			IF CIR_STOP_REQ THEN Pump_En[2] := 1;
			ELSIF CIR_RUN_REQ THEN Pump_En[2] := 0;
			ELSE Pump_En[2] := BOOL_TO_WORD(NOT Delay.OUT);
			END_IF

			(* Set RUN signal (for external objects) *)
			IF AlarmCtr>0 THEN (*OR fPump_ST[1].OUT OR fPump_ST[2].OUT THEN*)
				Run:=FALSE;
			ELSE
				Run:=SEL(Pump_En[2]=1,FALSE,TRUE);
			END_IF
		END_IF


	1,2:  (*** Alternate working and Master/backup mode ***)
		IF fCIR_AUTO[ActivePump].IN THEN
			(* If priority request *)
			IF CIR_STOP_REQ THEN Pump_En[ActivePump] := 1;
			ELSIF CIR_RUN_REQ THEN Pump_En[ActivePump] := 0;
			ELSE Pump_En[ActivePump] := BOOL_TO_WORD(NOT Delay.OUT);
			END_IF

			fBackup(IN:=(AlarmHw[ActivePump].OUT));

			IF fBackup.EVH THEN
				ActivePump := SEL(ActivePump=1,1,2);
				LogEv(EL_Wrn,EO_CIRD,ID,16,'');	(* Pump switched because of current pump failure *)

				(* Switch off old active pump *)
				IF ActivePump=1 THEN Pump_En[2] := 1;
				ELSE Pump_En[1] := 1;
				END_IF
			END_IF


			(* Set RUN signal (for external objects) *)
			IF AlarmCtr>0 THEN (*OR fPump_ST[ActivePump].OUT THEN*)
				Run:=FALSE;
			ELSE
				IF (ActivePump=1 AND PumpB_AUTO) OR (ActivePump=2 AND PumpA_AUTO) THEN
					Run:=SEL(Pump_En[ActivePump]=1,TRUE,FALSE);
				END_IF
			END_IF

		END_IF

END_CASE

(* Check if a pump enable update (modbus write) is requested *)
fPump_En[1](IN:=(Pump_En[1]=1));
fPump_En[2](IN:=(Pump_En[2]=1));

IF fPump_En[1].EVH OR fPump_En[1].EVL THEN
	Refresh_Now := TRUE;
END_IF

IF fPump_En[2].EVH OR fPump_En[2].EVL THEN
	Refresh_Now := TRUE;
END_IF
END_ACTION
ACTION Stm:
CASE state OF
	0:	(* Refresh time manager *)
		ReadTmr(IN:=NOT ReadTmr.Q);
		TimeOutModBus(In:=state<>0,PT:=t#5s);
		IF (ReadTmr.Q AND NodoDaInterrogare=Address1 )OR Refresh_Now AND NOT InibiscoModbus THEN
			state := 10;
			ReadTmr.PT := T#10s;  (* moreno *)
			InibiscoModbus := TRUE;
			Refresh_Now := FALSE;
		END_IF

	(**** READ CIR PARAMETERS ****)

	(**** PUMP 1 ****)
	10:	(* richiedo lettura stato Pompa  *)

			Modbus.MB_Query.SlaveAddress := Address1;
			Modbus.MB_Query.FunctionCode := 3;
			ModBus.MB_Query.Read_StartAddress := 201;
			ModBus.MB_Query.Read_Quantity := 2;
			ModBus.MB_Start := TRUE;

			state := 20;

	20:	(* Ripsosta *)
		IF NOT ModBus.MB_Start   THEN

			VerificaFuctionCode:=ModBus.MB_Resp.FunctionCode;
			VerificaNodoLetto:=ModBus.MB_Resp.SlaveAddress;
			IF ModBus.MB_MASTER.MB_Error<>0 THEN
				state := 45;
			ELSE
				DataPump1.PumpStatus := ModBus.MB_Resp.Data[0];
				DataPump1.PumpFault	:= WORD_TO_BOOL(ModBus.MB_Resp.Data[1]);

				Modbus.MB_Query.SlaveAddress := Address1;
				Modbus.MB_Query.FunctionCode := 3;
				ModBus.MB_Query.Read_StartAddress := 210;
				ModBus.MB_Query.Read_Quantity := 12;
				ModBus.MB_Start := TRUE;

				state := 30;
			END_IF
		END_IF

	30: (* Ripsota Altri paramenti Stato Pompa *)
		IF NOT ModBus.MB_Start  THEN

			IF ModBus.MB_MASTER.MB_Error<>0 THEN (*OR ModBus.MB_MASTER.MB_Error<>0 THEN*)
				state := 45;
			ELSE
				DataPump1.PumpBoardTemp 	:= WORD_TO_INT(ModBus.MB_Resp.Data[0]);
				DataPump1.PumpVoltage	:= ModBus.MB_Resp.Data[2];
				DataPump1.PumpCurrent	:= ModBus.MB_Resp.Data[3];
				DataPump1.PumpRPM		:= ModBus.MB_Resp.Data[5];
				DataPump1.PumpPower		:= ModBus.MB_Resp.Data[6];
				DataPump1.PumpOpTime		:= BUILD_16TO32(ADR(ModBus.MB_Resp.Data[7]));
				DataPump1.PumpHead		:= ModBus.MB_Resp.Data[9];
				DataPump1.PumpFlow		:= ModBus.MB_Resp.Data[10];
				DataPump1.PumpLiqTemp	:= WORD_TO_INT(ModBus.MB_Resp.Data[11]);


				ModBus.MB_Query.Read_StartAddress := 230; (* Lettura Allarmi presenti nella pompa *)
				ModBus.MB_Query.Read_Quantity := 1;(*15;*)
				ModBus.MB_Start := TRUE;

				state := 40;
			END_IF
		END_IF

	40:	(* Read alarms *)
		IF NOT ModBus.MB_Start   THEN
			IF ModBus.MB_MASTER.MB_Error<>0 THEN (*OR ModBus.MB_MASTER.MB_Error<>0 THEN*)
				state := 45;
			ELSE
				DataPump1.PumpAlarm[0] := ModBus.MB_Resp.Data[0];	(* Read just last (most recent) alarm *)
				(*DataPump.PumpAlarm[1] := ModBus.MB_Resp.Data[1];
				DataPump.PumpAlarm[2] := ModBus.MB_Resp.Data[2];
				DataPump.PumpAlarm[3] := ModBus.MB_Resp.Data[3];
				DataPump.PumpAlarm[4] := ModBus.MB_Resp.Data[4];
				DataPump.PumpAlarm[5] := ModBus.MB_Resp.Data[5];
				DataPump.PumpAlarm[6] := ModBus.MB_Resp.Data[6];
				DataPump.PumpAlarm[7] := ModBus.MB_Resp.Data[7];
				DataPump.PumpAlarm[8] := ModBus.MB_Resp.Data[8];
				DataPump.PumpAlarm[9] := ModBus.MB_Resp.Data[9];
				DataPump.PumpAlarm[10] := ModBus.MB_Resp.Data[10];
				DataPump.PumpAlarm[11] := ModBus.MB_Resp.Data[11];
				DataPump.PumpAlarm[12] := ModBus.MB_Resp.Data[12];
				DataPump.PumpAlarm[13] := ModBus.MB_Resp.Data[13];
				DataPump.PumpAlarm[14] := ModBus.MB_Resp.Data[14];*)

				state := 41;

			END_IF
		END_IF

(**** Dopo La Lettura Scrivo i paramentri ON/OFF e la velocità  ****)
	 41:	(* Scrivo il comando alla pompa A *)

		Modbus.MB_Query.SlaveAddress := Address1;
		Modbus.MB_Query.FunctionCode := 16;
		ModBus.MB_Query.Write_StartAddress := 109;
		ModBus.MB_Query.Write_Quantity :=2;
		ModBus.MB_Query.Write_Data[0] := VelocitaRichiesta;
		ModBus.MB_Query.Write_Data[1] := Pump_En[1];
		ModBus.MB_Start := TRUE;

		state := 42;

	42:	(* Read alarms *)
		IF NOT ModBus.MB_Start   THEN
			IF ModBus.MB_MASTER.MB_Error<>0 THEN (*OR ModBus.MB_MASTER.MB_Error<>0 THEN*)
				state := 45;
			ELSE
				state := 50;
			END_IF
		END_IF


	(**** CHECK MODBUS ERROR ****)
	45: 	(* Release MODBUS *)
			MODBUS.MB_Lock:=FALSE;

			(* Retries *)
			retry:=retry+1;
			IF retry>3 THEN
				retry:=0;
				(* Verify if slave is dead *)
				IF retryErr < retryErrMaX THEN
					retryErr := retryErr + 1;
				ELSE
					fModbusAlr := TRUE;
					(* Verify ModBus error	*)

					IF fModbusAlr AND ErroreComuModBus1=FALSE THEN
						LogEv(EL_Alarm,EO_CIRDM,ID,13,CONCAT('ErroreModbus_',INT_TO_STRING(ModBus.MB_MASTER.MB_Error)));
						ErroreComuModBus1 := TRUE;
					END_IF
					IF fModbusAlr=FALSE AND retryErr=0 THEN
						LogEv(EL_Log,EO_CIRDM,ID,14,'ComunicazioneModBus_OK');
							ErroreComuModBus1 := FALSE;
					(*	WarningCtr := SEL(WarningCtr=0, WarningCtr-1, 0); *)
					END_IF
				END_IF
				Refresh_Now := FALSE;
			END_IF

			state:=50;



	(**** PUMP 2 ****)
	50:	(* richiedo lettura stato Pompa  *)

			Modbus.MB_Query.SlaveAddress := Address2;
			Modbus.MB_Query.FunctionCode := 3;
			ModBus.MB_Query.Read_StartAddress := 201;
			ModBus.MB_Query.Read_Quantity := 2;
			ModBus.MB_Start := TRUE;

			state := 60;

	60:	(* Ripsosta *)
		IF NOT ModBus.MB_Start   THEN

			VerificaFuctionCode:=ModBus.MB_Resp.FunctionCode;
			VerificaNodoLetto:=ModBus.MB_Resp.SlaveAddress;
			IF ModBus.MB_MASTER.MB_Error<>0 THEN
				state := 300;
			ELSE
				DataPump2.PumpStatus := ModBus.MB_Resp.Data[0];
				DataPump2.PumpFault	:= WORD_TO_BOOL(ModBus.MB_Resp.Data[1]);

				Modbus.MB_Query.SlaveAddress := Address2;
				Modbus.MB_Query.FunctionCode := 3;
				ModBus.MB_Query.Read_StartAddress := 210;
				ModBus.MB_Query.Read_Quantity := 12;
				ModBus.MB_Start := TRUE;

				state := 70;
			END_IF
		END_IF

	70: (* Ripsota Altri paramenti Stato Pompa *)
		IF NOT ModBus.MB_Start  THEN

			IF ModBus.MB_MASTER.MB_Error<>0 THEN (*OR ModBus.MB_MASTER.MB_Error<>0 THEN*)
				state := 300;
			ELSE
				DataPump2.PumpBoardTemp 	:= WORD_TO_INT(ModBus.MB_Resp.Data[0]);
				DataPump2.PumpVoltage	:= ModBus.MB_Resp.Data[2];
				DataPump2.PumpCurrent	:= ModBus.MB_Resp.Data[3];
				DataPump2.PumpRPM		:= ModBus.MB_Resp.Data[5];
				DataPump2.PumpPower		:= ModBus.MB_Resp.Data[6];
				DataPump2.PumpOpTime		:= BUILD_16TO32(ADR(ModBus.MB_Resp.Data[7]));
				DataPump2.PumpHead		:= ModBus.MB_Resp.Data[9];
				DataPump2.PumpFlow		:= ModBus.MB_Resp.Data[10];
				DataPump2.PumpLiqTemp	:= WORD_TO_INT(ModBus.MB_Resp.Data[11]);


				ModBus.MB_Query.Read_StartAddress := 230; (* Lettura Allarmi presenti nella pompa *)
				ModBus.MB_Query.Read_Quantity := 1;(*15;*)
				ModBus.MB_Start := TRUE;

				state := 80;
			END_IF
		END_IF

	80:	(* Read alarms *)
		IF NOT ModBus.MB_Start   THEN
			IF ModBus.MB_MASTER.MB_Error<>0 THEN (*OR ModBus.MB_MASTER.MB_Error<>0 THEN*)
				state := 300;
			ELSE
				DataPump2.PumpAlarm[0] := ModBus.MB_Resp.Data[0];	(* Read just last (most recent) alarm *)
				(*DataPump.PumpAlarm[1] := ModBus.MB_Resp.Data[1];
				DataPump.PumpAlarm[2] := ModBus.MB_Resp.Data[2];
				DataPump.PumpAlarm[3] := ModBus.MB_Resp.Data[3];
				DataPump.PumpAlarm[4] := ModBus.MB_Resp.Data[4];
				DataPump.PumpAlarm[5] := ModBus.MB_Resp.Data[5];
				DataPump.PumpAlarm[6] := ModBus.MB_Resp.Data[6];
				DataPump.PumpAlarm[7] := ModBus.MB_Resp.Data[7];
				DataPump.PumpAlarm[8] := ModBus.MB_Resp.Data[8];
				DataPump.PumpAlarm[9] := ModBus.MB_Resp.Data[9];
				DataPump.PumpAlarm[10] := ModBus.MB_Resp.Data[10];
				DataPump.PumpAlarm[11] := ModBus.MB_Resp.Data[11];
				DataPump.PumpAlarm[12] := ModBus.MB_Resp.Data[12];
				DataPump.PumpAlarm[13] := ModBus.MB_Resp.Data[13];
				DataPump.PumpAlarm[14] := ModBus.MB_Resp.Data[14];*)

				state := 100;

			END_IF
		END_IF


	(**** Dopo La Lettura Scrivo i paramentri ON/OFF e la velocità  ****)
	 100:	(* Scrivo il comando alla pompa A *)

		Modbus.MB_Query.SlaveAddress := Address1;
		Modbus.MB_Query.FunctionCode := 16;
		ModBus.MB_Query.Write_StartAddress := 109;
		ModBus.MB_Query.Write_Quantity :=2;
		ModBus.MB_Query.Write_Data[0] := VelocitaRichiesta;
		ModBus.MB_Query.Write_Data[1] := Pump_En[1];
		ModBus.MB_Start := TRUE;

		state := 110;


		110: (* Scrivo il comando alla pompa B *)
		IF NOT ModBus.MB_Start THEN
			IF ModBus.MB_MASTER.MB_Error<>0 THEN (*OR ModBus.MB_MASTER.MB_Error<>0 THEN*)
				state := 300;
			ELSE
				Modbus.MB_Query.SlaveAddress := Address2;
				Modbus.MB_Query.FunctionCode := 16;
				ModBus.MB_Query.Write_StartAddress := 109;
				ModBus.MB_Query.Write_Quantity :=2;
				ModBus.MB_Query.Write_Data[0] := VelocitaRichiesta;
				ModBus.MB_Query.Write_Data[1] := Pump_En[2];
				ModBus.MB_Start := TRUE;

			state := 120;
			END_IF
		END_IF


		120:
		IF NOT ModBus.MB_Start THEN
			IF ModBus.MB_MASTER.MB_Error<>0 THEN (*OR ModBus.MB_MASTER.MB_Error<>0 THEN*)
				state := 300;
			ELSE
				IF fModbusAlr THEN fModbusAlr := FALSE; END_IF

				NodoDaInterrogare:=Address2+1; (* qui il passo è doppio *)
				InibiscoModbus:=FALSE;
				retryErr := 0;
				retry := 0;
				state := 0;
			END_IF
		END_IF



	(**** CHECK MODBUS ERROR ****)
	300: 	(* Release MODBUS *)
			MODBUS.MB_Lock:=FALSE;

			(* Retries *)
			retry:=retry+1;
			IF retry>3 THEN
				retry:=0;
				(* Verify if slave is dead *)
				IF retryErr < retryErrMaX THEN
					retryErr := retryErr + 1;
				ELSE
					fModbusAlr := TRUE;
					(* Verify ModBus error	*)

					IF fModbusAlr AND ErroreComuModBus2=FALSE THEN
						LogEv(EL_Alarm,EO_CIRDM,ID,13,CONCAT('ErroreModbus_',INT_TO_STRING(ModBus.MB_MASTER.MB_Error)));
						ErroreComuModBus2 := TRUE;
					END_IF
					IF fModbusAlr=FALSE AND retryErr=0 THEN
						LogEv(EL_Log,EO_CIRDM,ID,14,'ComunicazioneModBus_OK');
							ErroreComuModBus2 := FALSE;
					(*	WarningCtr := SEL(WarningCtr=0, WarningCtr-1, 0); *)
					END_IF
				END_IF


				Refresh_Now := FALSE;
			END_IF

			NodoDaInterrogare:=Address2+1; (* qui il passo è doppio *)
			state:=0;
END_CASE



(* Controllo Time Out Ciclo ModBus *)

TimeOutModBus(In:=state<>0,PT:=t#5s);
IF TimeOutModBus.Q THEN
	State:=0;
	Refresh_Now:=TRUE;  (* Rilancio la lettura del nodo *)
	IF MODBUS.MB_Lock=TRUE THEN MODBUS.MB_Lock:=FALSE;END_IF
	IF InibiscoModbus=TRUE THEN InibiscoModbus:=FALSE;END_IF
END_IF
END_ACTION

(* POU Plant_Objects/obj_MODBUS_TCP, ST *)
FUNCTION_BLOCK obj_MODBUS_TCP
(* === MODBUS-TCP PROTOCOL INTERFACE ===
   v1.0[10/06/15] - Create
*)
VAR CONSTANT
	VARS_Max	: BYTE := 32;
END_VAR
VAR_INPUT
	(* Settings *)
	ID			: BYTE;
	IP			: STRING;
	PORT		: WORD:=502;
	(* Interface *)
	MB_MASTER	: ETHERNET_MODBUSMASTER_TCP;
	MB_READBUF	: ARRAY [0..128] OF WORD;
	MB_WRITEBUF : ARRAY [0..128] OF WORD;
	MB_Start	: BOOL;
	MB_Lock		: BOOL;
	(* Variables management *)
	VARS_En		: BOOL;
	VARS		: ARRAY [0..VARS_Max] OF typ_MODBUS_VAR;
	VARS_Check	: BOOL;
	VARS_Alarm	: BOOL;
	(* Variables allocation *)
	VAR_Pointer : POINTER TO ARRAY[0..99] OF WORD;
	VAR_Cfg		: POINTER TO typ_MODBUS_VAR;
END_VAR
VAR_OUTPUT
	(* Status *)
	Status_Log	: BYTE;
	Status_Vis	: DWORD;
END_VAR
VAR
	sta         : BYTE :=0;
	i			: BYTE;
	j			: BYTE;
	Alarm		: FLT_EVENT;

	VarTmr		: TON := (PT:=T#1s);
	VarSta		: BYTE; (* Status *)
	VarCnt		: BYTE; (* Scan counter *)
	VarRetry	: BYTE;
	VarAlarm	: BYTE; (* Last variable with errors *)
END_VAR
MB_MASTER( strIP_ADDRESS:=IP, wPORT:=PORT, tTIME_OUT:=T#750MS, (*xCONNECT:=TRUE,*)
		   ptREAD_DATA:=ADR(MB_READBUF), ptSEND_DATA:=ADR(MB_WRITEBUF), xSEND:=MB_Start );

IF sta=0 THEN
	MB_MASTER.xCONNECT:=TRUE;
	sta:=1;
END_IF

(* Process variable management *)
IF VARS_En THEN VARS_Process(); END_IF

(* Check status *)
Alarm(IN:=(MB_MASTER.wERROR<>0));
IF Alarm.EVH THEN
	LogEv(SEL(MB_MASTER.wERROR>0,EL_Wrn,EL_Alarm),EO_MODBUS_TCP,ID,1,WORD_TO_STRING(MB_MASTER.wERROR));
END_IF
IF Alarm.EVL THEN
	LogEv(EL_Log,EO_MODBUS_TCP,ID,2,'');
END_IF

(* Log/visu status *)
   IF Alarm.IN   THEN Status_Log:=2; Status_Vis:=COLOR_RED;
ELSIF Vars_Alarm THEN Status_Log:=1; Status_Vis:=COLOR_YELLOW;
  				 ELSE Status_Log:=0; Status_Vis:=COLOR_GREEN;
END_IF
END_FUNCTION_BLOCK
ACTION VAR_Search:
(* Search VAR with specific pointer if not found return first free VAR
	[Last VAR is not active... used as safe area...] 
*)
j:=VARS_Max;
FOR i := 0 TO VARS_Max-1 DO
	IF VARS[i].Variable=0 AND j>i THEN j:=i; END_IF
	IF VARS[i].Variable=VAR_Pointer THEN
		VAR_Cfg:=ADR(VARS[i]);
		RETURN;
	END_IF
END_FOR
VAR_Cfg:=ADR(VARS[j]);
END_ACTION
ACTION VARS_Process:
(* Update var timers *)
VarTmr(IN:=(NOT VarTmr.Q));
IF VarTmr.Q THEN
	FOR i := 0 TO VARS_Max DO
		IF VARS[i].Refresh_Cnt>0 THEN VARS[i].Refresh_Cnt:=VARS[i].Refresh_Cnt-1; END_IF
	END_FOR
	VARS_Check:=TRUE;
END_IF


(* Process status *)
CASE VarSta OF
	0: (* === Init *)
		VarCnt:=0;
		VarSta:=1;

	1: (* === Wait check signal *)
		IF VARS_Check THEN
			VARS_Check:=FALSE;
			VarCnt:=0;
			VarSta:=2;
		END_IF

	2: (* === Check loop *)
		IF NOT (MB_Lock OR MB_Start) THEN
			WHILE VarCnt<=(VARS_Max-1) AND VarSta=2 DO
				(* Check only active vars *)
				IF VARS[VarCnt].Variable<>0 THEN
					(* Check var auto-refresh on timer checks *)
					IF VARS[VarCnt].Refresh_Time>0 AND VARS[VarCnt].Refresh_Cnt=0 THEN
						VARS[VarCnt].Refresh_Cnt:=VARS[VarCnt].Refresh_Time;
						VarSta:=3;
					END_IF
					(* Check refresh for change or request *)
					CASE VARS[VarCnt].FunCode OF
						5,6,15,16: (* Write functions *)
							IF VARS[VarCnt].Variable_Size=1 THEN
								IF VARS[VarCnt].Variable^<>VARS[VarCnt].Variable_Mirror THEN
									VARS[VarCnt].Variable_Mirror:=VARS[VarCnt].Variable^;
									VarSta:=3;
								END_IF
							ELSE
								IF VARS[VarCnt].Variable_Mirror<>0 THEN
									VARS[VarCnt].Variable_Mirror:=0;
									VarSta:=3;
								END_IF
							END_IF
						1,2,3,4: (* Write functions *)
							IF VARS[VarCnt].Variable_Mirror<>0 THEN
								VARS[VarCnt].Variable_Mirror:=0;
								VarSta:=3;
							END_IF
					END_CASE
				END_IF
				(* Process query *)
				IF VarSta=3 THEN
					MB_Lock:=TRUE;
					MB_MASTER.bUNIT_ID:=VARS[VarCnt].SlaveAddress;
					MB_MASTER.bFUNCTION_CODE:=VARS[VarCnt].FunCode;
					CASE VARS[VarCnt].FunCode OF
						16#5,16#6,16#F,16#10:
							MB_MASTER.wREAD_ADDRESS:=0;
							MB_MASTER.wREAD_QUANTITY:=0;
							MB_MASTER.wWRITE_ADDRESS:=VARS[VarCnt].FunAddress;
							MB_MASTER.wWRITE_QUANTITY:=VARS[VarCnt].Variable_Size;
							IF VARS[VarCnt].Variable_Size=200 THEN
								COPY_32SWAP16(VARS[VarCnt].Variable, ADR(MB_WRITEBUF));
							ELSIF VARS[VarCnt].Variable_Size>1 THEN
								MEMCPY(VARS[VarCnt].Variable, ADR(MB_WRITEBUF), 2*VARS[VarCnt].Variable_Size);
							ELSE
								MB_WRITEBUF[0]:=VARS[VarCnt].Variable^;
							END_IF
						16#1,16#2,16#3,16#4:
							MB_MASTER.wREAD_ADDRESS:=VARS[VarCnt].FunAddress;
							IF VARS[VarCnt].Variable_Size=200 THEN MB_MASTER.wREAD_QUANTITY:=2; ELSE
							  MB_MASTER.wREAD_QUANTITY:=VARS[VarCnt].Variable_Size;
							END_IF
							MB_MASTER.wWRITE_ADDRESS:=0;
							MB_MASTER.wWRITE_QUANTITY:=0;
					END_CASE
					VarRetry:=0;
					MB_Start:=TRUE;
				ELSE
					VarCnt:=VarCnt+1;
				END_IF
			END_WHILE
			(* Check loop completed -> no actions *)
			IF VarSta=2 THEN VarSta:=1; END_IF
		END_IF

	3: (* === Wait & process MB response *)
		IF NOT MB_Start THEN
			IF MB_MASTER.wERROR=0 THEN
				CASE VARS[VarCnt].FunCode OF
					1,2,3,4:
						IF VARS[VarCnt].Variable_Size=200 THEN
							COPY_32SWAP16(ADR(MB_READBUF), VARS[VarCnt].Variable);
						ELSIF VARS[VarCnt].Variable_Size>1 THEN
							MEMCPY(ADR(MB_READBUF), VARS[VarCnt].Variable, 2*VARS[VarCnt].Variable_Size);
						ELSE
							VARS[VarCnt].Variable^:=MB_READBUF[0];
						END_IF
				END_CASE
				MB_Lock:=FALSE;
				(* Signal error recovery *)
				IF VARS_Alarm=TRUE AND VarCnt=VarAlarm THEN
					LogEv(EL_Wrn,EO_MODBUS_TCP,ID,5,'');
					VARS_Alarm:=FALSE;
				END_IF
				(* Next var *)
				VarCnt:=VarCnt+1;
				VarSta:=2;
			ELSE
				IF VarRetry<10 THEN
					VarRetry:=VarRetry+1;
					MB_Start:=TRUE;
				ELSE
					MB_Lock:=FALSE;
					(* Signal error *)
					IF VARS_Alarm=FALSE THEN
						LogEv(EL_Wrn,EO_MODBUS_TCP,ID,3,WORD_TO_STRING(MB_MASTER.wERROR));
						VARS_Alarm:=TRUE;
						VarAlarm:=VarCnt-1;
					END_IF
					(* Next var *)
					VarCnt:=VarCnt+1;
					VarSta:=2;
				END_IF
			END_IF
		END_IF

ELSE
	VarSta:=0;
END_CASE
END_ACTION

(* POU Plant_Objects/obj_TPV, ST *)
FUNCTION_BLOCK obj_TPV
(* === TEMPERATURE PROBE  ===
   v1.0[16/04/15] - Versioning
*)
VAR CONSTANT
	NormalEv		: BYTE := 0;
	ErrorEv			: BYTE := 1;
	WarningEv		: BYTE := 2;
END_VAR
VAR_INPUT
	(* Settings *)
	ID				: BYTE;
	TAP				: BYTE:=4;	   (* Consecutive checks filter *)
	INITEV			: BOOL:= TRUE; (* Generate init OK event *)
	IN_EMIN			: INT :=-2000; (* Low error limit *)
	IN_WMIN			: INT := -550; (* Low warning value *)
	IN_WMAX			: INT :=  900; (* High warning value *)
	IN_EMAX			: INT := 8500; (* High error limit *)
	ERR_MIN_SHORT	: BOOL:= TRUE; (* TRUE  ==> EMIN=Short        , EMAX=Disconnected
									  FALSE ==> EMIN=Disconnected , EMAX=Short 		 *)
	(* Physical input *)
	IN			: INT;
END_VAR
VAR_OUTPUT
	WRN			: BOOL;	(* Value in warning range *)
	ERR			: BOOL;	(* Value error *)
	HI			: INT;	(* Highest value - cleared by Stat_Reset() action *)
	AVG			: INT; 	(* Average value - updated by Mean() action, cleared by Mean_Reset() action *)
	LOW			: INT;	(* Lowest value  - cleared by Stat_Reset() action *)

	Status_Log	: WORD;
	Status_Vis	: DWORD;
END_VAR
VAR
	cnt			: BYTE;
	event		: BYTE := 0;	(* 0: monitoring a generic, 1: monitoring an error, 2: monitoring a warning *)
	asum		: DINT;
	acnt		: WORD;
END_VAR
(* Check probe value limits *)
IF IN<=IN_EMIN OR IN>=IN_EMAX THEN
	IF NOT ERR THEN
		IF event <> ErrorEv THEN
			cnt := 1;
			event := ErrorEv;
		ELSE
			cnt:=cnt+1;
		END_IF

		IF cnt>TAP THEN
			cnt:=0;
			ERR:=TRUE; WRN:=FALSE;
			IF ( ERR_MIN_SHORT=TRUE  AND IN<=IN_EMIN ) OR ( ERR_MIN_SHORT=FALSE AND IN>=IN_EMAX ) THEN
				LogEv(EL_Alarm,EO_TPV,ID,5,INT_TO_STRING(IN));
			ELSE
				LogEv(EL_Alarm,EO_TPV,ID,4,INT_TO_STRING(IN));
			END_IF
		END_IF
	END_IF
ELSIF IN<=IN_WMIN OR IN>=IN_WMAX THEN
	IF NOT WRN THEN
		IF event <> WarningEv THEN
			cnt := 1;
			event := WarningEv;
		ELSE
			cnt:=cnt+1;
		END_IF

		IF cnt>TAP THEN
			cnt:=0;
			ERR:=FALSE; WRN:=TRUE;
			LogEv(EL_Wrn,EO_TPV,ID,SEL(IN<=IN_WMIN,3,2),INT_TO_STRING(IN));
		END_IF
	END_IF
ELSE
	IF INITEV OR WRN OR ERR THEN
		IF event <> NormalEv THEN
			cnt := 1;
			event := NormalEv;
		ELSE
			cnt:=cnt+1;
		END_IF

		IF cnt>TAP THEN
			cnt:=0;
			INITEV:=FALSE; ERR:=FALSE; WRN:=FALSE;
			LogEv(EL_Log,EO_TPV,ID,1,'Probe_OK');
		END_IF
	END_IF
END_IF
(*
(* Average value *)
IF acnt>=500 THEN
	Mean();
	asum := asum - AVG;
	acnt := acnt - 1;
END_IF

asum := asum + IN;
acnt := acnt + 1;
*)
AVG := IN;


(* Statistics values *)
IF IN<LOW THEN LOW:=IN; END_IF
IF IN>HI  THEN HI :=IN; END_IF



(* Status Log *)
IF ERR THEN	Status_Log := 2; Status_Vis := COLOR_RED;
ELSIF WRN THEN Status_Log := 1;	Status_Vis := COLOR_YELLOW;
ELSE Status_Log := 0; Status_Vis := COLOR_GREEN;
END_IF
END_FUNCTION_BLOCK
ACTION AddLogData:
Logger.s1:=INSERT('&TPV=',BYTE_TO_STRING(ID),4);
IF ID<10 THEN Logger.s1:=INSERT(Logger.s1,'0',4); END_IF



Logger.s1:=CONCAT(Logger.s1,INT_TO_STRING(AVG));		Logger.s1:=CONCAT(Logger.s1,';');

Logger.s1:=CONCAT(Logger.s1,WORD_TO_STRING(Status_Log));
ADDSTRING(ADR(Logger.TData), ADR(Logger.s1), Logger.TLen);
END_ACTION
ACTION Mean:
AVG := DINT_TO_INT(asum/acnt);
END_ACTION
ACTION Mean_Reset:
AVG:=IN;
asum:=IN;
acnt:=1;
END_ACTION
ACTION Stat_Reset:
HI:=IN;
LOW:=IN;
END_ACTION

(* POU Plant_Objects/obj_VRD_new, ST *)
FUNCTION_BLOCK obj_VRD_new
(* === VALVOLA RIPARTITORE ===
   v1.0[16/04/15] - Versioning
*)
VAR CONSTANT
	Chk_CntSecAlarm	: INT := 900;	(* 900s = 15 minutes -> Observation itme *)
END_VAR
VAR_INPUT
	(* Settings *)
	ID				: BYTE;
	(* Controls *)
	RUN  			: BOOL;					(* Control input *)
	ReducedRange	: BOOL := FALSE;		(* If true output value is among 2 and 10V, otherwise 0-10V *)

	(* Physical inputs *)
	TEMP 			: INT;		(* Input temperature from sensor *)
	STATUS 			: WORD;		(* Input position from valve *)

	InitOK			: BOOL;
	Alarm1			: BOOL;
	Alarm2			: BOOL;
	Warning			: BOOL;

	Ctrl_Init		: BOOL;
	Ctrl_SetPoint	: INT;
	Ctrl_SetPointNew: INT := 0;
	Delta_SetPoint	: INT;
	Ctrl_Err		: INT;			(* Current error *)
	Ctrl_Err0		: INT; 			(* Previous error *)
	Ctrl_Accel		: REAL;			(* Derivate of error *)
	Ctrl_AccelGate  : INT:=1;		(* Derivate gate *)
	Ctrl_AccelTmr	: WORD;
	Ctrl_SetPointGate: INT := 5;	(* Setpoint gate - 0.5°C *)
	Ctrl_ErrGate	: INT:=5;		(* Error gate *)
	Ctrl_Kp			: REAL:=2;(*1;*)		(* Proportional factor *)
	Ctrl_Kd			: REAL:=10;(*100;*)  	(* Derivative factor *)
	Ctrl_Out		: REAL;

	Chk_Err			: INT;
	Chk_ErrGate		: INT:=20; 		(* Check error gate *)
	Chk_Cnt			: INT;
	Chk_CntAlarm	: INT:=240; 		(* Check error trigger 120s *)

	(* Status *)
	Log_AvgTemp		: AVERAGE_T;
	Status_Log		: BYTE;
	Status_Vis 		: DWORD;

	(* Feedback *)
	fFeedback		: BOOL;			(* TRUE: Feedback available, FALSE: Feedback not available *)

	OffsetBoost: INT;
END_VAR
VAR_IN_OUT
	CLIM		: typ_Clima;
END_VAR
VAR_OUTPUT
	(* Physical outputs *)
	OUT			: WORD;
END_VAR
VAR
	Curve		: CHARCURVE;
	Curve_Err	: BYTE;

	aTemp		: ARRAY [1..20] OF INT;
	meanTemp	: INT;
	sum			: INT := 0;
	Tmr			: TON := (PT:=T#1s);
	index		: BYTE;
	i			: BYTE;
	fCtrl_Err	: BOOL;		(* TRUE: Ctrl_Err>0, FALSE: Ctrl_Err<0 *)

END_VAR
(* Check initialization *)
(*IF NOT InitOK THEN Init(); END_IF*)

(* Check max temperature *)
IF TEMP>Plant_VRD_TAlarm THEN
	IF NOT Alarm1 THEN
		Alarm1:=TRUE;
		LogEv(EL_AlarmStop,EO_VRD,ID,3,'VRD_Overtemperature');
	END_IF
END_IF

(* Check climatic setup *)
IF NOT CLIM.InitOK THEN	DefaultClim(); END_IF;
(* Calculate Setpoint *)
Curve(	IN:= T_AMB,	N:= 5, P:= CLIM.Points,			(* Given the x value as input, the corresponding y value as output is returned, if it matches the crve designed by array of points *)
		OUT=> Ctrl_SetPointNew, ERR=> Curve_Err );

Ctrl_SetPointNew:=Ctrl_SetPointNew+OffsetBoost;

IF Curve_Err>0 OR Ctrl_SetPoint>Plant_VRD_TMax THEN
	Ctrl_SetPoint:=Plant_VRD_TDefault;
	IF NOT Warning THEN
		Warning:=TRUE;
		LogEv(EL_Wrn,EO_VRD,ID,2,'VRD_Climatic_Error');
	END_IF
ELSE
	Delta_SetPoint := ABS(Ctrl_SetPoint - Ctrl_SetPointNew);
	IF Delta_SetPoint>Ctrl_SetPointGate THEN Ctrl_SetPoint := Ctrl_SetPointNew; END_IF

	Warning:=FALSE;
END_IF

(* Execute control loop [T=500ms] *)
IF RUN AND (NOT Alarm1) THEN
	(* Calculate error *)
	Ctrl_Err:=Ctrl_SetPoint-TEMP;
	(* Init/restart operations *)
	IF NOT Ctrl_Init THEN
		Ctrl_Accel:=0;
		Ctrl_AccelTmr:=0;
		Ctrl_Err0:=Ctrl_Err;
		Ctrl_Out:=5000;
		Ctrl_Init:=TRUE;
	END_IF
	(* Calculate acceleration *)
	IF ABS(Ctrl_Err-Ctrl_Err0)>Ctrl_AccelGate OR Ctrl_AccelTmr>20 THEN
		Ctrl_Accel:=INT_TO_REAL(Ctrl_Err-Ctrl_Err0)/WORD_TO_REAL(1+Ctrl_AccelTmr);
		Ctrl_AccelTmr:=0;
		Ctrl_Err0:=Ctrl_Err;
	ELSE
		Ctrl_AccelTmr:=Ctrl_AccelTmr+1;
	END_IF

	(* Gate error *)
	IF ABS(Ctrl_Err)>Ctrl_ErrGate THEN
		(* Control loop *)
		Ctrl_Out:=Ctrl_Out+(Ctrl_Kp*Ctrl_Err)+(Ctrl_Kd*Ctrl_Accel);
	END_IF

	(* Limiter and Output *)
	Ctrl_Out:=LIMIT(0,Ctrl_Out,32766);
	OUT:=REAL_TO_WORD(Ctrl_Out);

ELSE
	Ctrl_Init:=FALSE;
	OUT:=0;
END_IF

(* If there is an hardware feedback (such as 0-10V, potentiometer, ...) check it otherwise try to rebuild it *)
IF fFeedback THEN CheckFeedback();
ELSE BuildFeedback();
END_IF

(* Status temp *)
Log_AvgTemp(IN:=Temp);


(* Status color *)
   IF Alarm1 OR Alarm2 THEN Status_Log:=2; Status_Vis:=16#2020F0;
ELSIF Warning          THEN Status_Log:=1; Status_Vis:=16#20F0F0;
                       ELSE Status_Log:=0; Status_Vis:=SEL(RUN,16#006000,16#20F020);
END_IF
END_FUNCTION_BLOCK
ACTION AddLogData:
Logger.s1:=INSERT('&VRD=',BYTE_TO_STRING(ID),4);
IF ID<10 THEN Logger.s1:=INSERT(Logger.s1,'0',4); END_IF

Logger.s1:=CONCAT(Logger.s1,INT_TO_STRING(Ctrl_SetPoint));				Logger.s1:=CONCAT(Logger.s1,';');
Logger.s1:=CONCAT(Logger.s1,WORD_TO_STRING(OUT));						Logger.s1:=CONCAT(Logger.s1,';');

IF fFeedback THEN Logger.s1:=CONCAT(Logger.s1,WORD_TO_STRING(STATUS));
ELSE Logger.s1:=CONCAT(Logger.s1,'0');	(* Bypass *)
END_IF

Logger.s1:=CONCAT(Logger.s1,';');

Logger.s1:=CONCAT(Logger.s1,WORD_TO_STRING(Status_Log));
ADDSTRING(ADR(Logger.TData), ADR(Logger.s1), Logger.TLen);
END_ACTION
ACTION BuildFeedback:
(* Comparison is taken between actual temperature vs windowed mean value of last 20 temperature
   (check is carried out every second)	*)
IF RUN AND (NOT Alarm1) THEN

	IF Ctrl_Err>0 THEN
		IF NOT fCtrl_Err THEN index := 0; END_IF
		fCtrl_Err := TRUE;
	ELSE
		IF fCtrl_Err THEN index := 0; END_IF
		fCtrl_Err := FALSE;
	END_IF

	(* Temperature is lower than setpoint -->> Should increase *)
	Tmr(IN:=NOT Tmr.Q);

	IF Tmr.Q THEN

		IF index<21 THEN
			(* Fullfil temperature array *)
			aTemp[index] := TEMP;
			index := index + 1;

			IF index=20 THEN
				FOR i:=1 TO 20 BY 1 DO sum := sum + aTemp[i]; END_FOR
			END_IF
		ELSE
			(* Calculate mean value *)
			meanTemp := sum/20;

			IF (fCtrl_Err AND TEMP<meanTemp) OR (NOT fCtrl_Err AND TEMP>meanTemp) THEN

				IF Chk_Cnt>Chk_CntSecAlarm THEN
					IF NOT Alarm2 THEN
						Alarm2:=TRUE;
						LogEv(EL_Alarm,EO_VRD,ID,4,'VRD_Position_Error');
					END_IF
				ELSE
					Chk_Cnt := Chk_Cnt+1;
				END_IF

			ELSE
				(* Reset counter and alarm flag *)
				Chk_Cnt:=0;
				Alarm2:=FALSE;
			END_IF

			sum := 0;	(* Reset sum counter *)

			(* Shift array removing oldest value *)
			FOR i:=1 TO 20 BY 1 DO
				aTemp[i-1] := aTemp[i];
				sum := sum + aTemp[i];
			END_FOR

			aTemp[20] := TEMP;			(* Last temperature value is new one *)
			sum := sum + aTemp[20];		(* Update sum *)
		END_IF
	END_IF
END_IF
END_ACTION
ACTION CheckFeedback:
(* Calculate position error according to feedback *)
IF ReducedRange THEN
(* SETPOINT[2..10V]-STATUS[0..10V] *)
	IF OUT<=6553 THEN Chk_Err:=0; ELSE Chk_Err:=(OUT-6553)/262; END_IF
	Chk_Err:=(Chk_Err-STATUS)/327;
ELSE
(* SETPOINT[0..10V]-STATUS[0..10V] *)
	Chk_Err := OUT - STATUS;
END_IF

(* Check position error *)
IF ( ABS(Chk_Err)>Chk_ErrGate ) THEN
	IF Chk_Cnt>Chk_CntAlarm THEN
		IF NOT Alarm2 THEN
			Alarm2:=TRUE;
			LogEv(EL_Alarm,EO_VRD,ID,4,'VRD_Position_Error');
		END_IF
	ELSE
		Chk_Cnt:=Chk_Cnt+1;
	END_IF
ELSE
	Chk_Cnt:=0;
	Alarm2:=FALSE;
END_IF
END_ACTION
ACTION DefaultClim:
(*CLIM.Points[0].X:=-300; CLIM.Points[0].Y:=400;
CLIM.Points[1].X:=-50;  CLIM.Points[1].Y:=400;
CLIM.Points[2].X:= 200; CLIM.Points[2].Y:=200;
CLIM.Points[3].X:= 300; CLIM.Points[3].Y:=200;
CLIM.Points[4].X:= 500; CLIM.Points[4].Y:=200;*)
CLIM.Points[0].X:=-300; CLIM.Points[0].Y:=850;
CLIM.Points[1].X:=-50;  CLIM.Points[1].Y:=650;
CLIM.Points[2].X:= 100; CLIM.Points[2].Y:=400;
CLIM.Points[3].X:= 200; CLIM.Points[3].Y:=200;
CLIM.Points[4].X:= 500; CLIM.Points[4].Y:=200;
CLIM.InitOK:=TRUE;
LogEv(EL_Wrn,EO_VRD,ID,1,'Climatic_Default');
END_ACTION
ACTION Init:
(* End initialization *)
InitOK:=TRUE;
END_ACTION

(* POU Plant_Objects/obj_VRD_POT_new, ST *)
FUNCTION_BLOCK obj_VRD_POT_new
(* === VALVOLA RIPARTITORE ===
   v1.0[16/04/15] - Versioning
*)
VAR CONSTANT
	ValveOpenRes	: WORD := 16#07D0;
	ValveCloseRes	: WORD := 16#EC00;

	ValvePosCheck	: BYTE :=4;

	Chk_CntSecAlarm	: INT := 900;	(* 900s = 15 minutes -> Observation itme *)
END_VAR
VAR_INPUT
	(* Settings *)
	ID				: BYTE;
	(* Controls *)
	RUN  			: BOOL;		(* Control input *)

	(* Physical inputs *)
	TEMP 			: INT;		(* Input temperature from sensor *)
	STATUS 			: WORD;		(* Input position from valve *)

	InitOK			: BOOL;
	Alarm1			: BOOL;
	Alarm2			: BOOL;
	Warning			: BOOL;

	Ctrl_Init		: BOOL;
	Ctrl_SetPoint	: INT;
	Ctrl_SetPointNew: INT := 0;
	Delta_SetPoint	: INT;
	Ctrl_Err		: INT;			(* Current error *)
	Ctrl_Err0		: INT; 			(* Previous error *)
	Ctrl_Accel		: REAL;			(* Derivate of error *)
	Ctrl_AccelGate  : INT:=1;		(* Derivate gate - 0.1°C/500ms *)
	Ctrl_AccelTmr	: WORD;
	Ctrl_SetPointGate: INT := 5;	(* Setpoint gate - 0.5°C *)
	Ctrl_Out		: REAL;

	(*Chk_Err			: INT;	*)
	Chk_Err			: REAL;
	Chk_Cnt			: INT;
	Chk_CntAlarm	: INT:=60; 		(* Check error trigger 60s *)

	(* Status *)
	Log_AvgTemp		: AVERAGE_T;

	(* Control parameters *)
	Tpwm			: TIME := T#2s;

	(* Feedback *)
	fFeedback		: BOOL;			(* TRUE: Feedback available, FALSE: Feedback not available *)


	OffsetBoost: INT;

END_VAR
VAR_IN_OUT
	CLIM		: typ_Clima;
END_VAR
VAR_OUTPUT
	(* Physical outputs *)
	OUT_CL		: BOOL;
	OUT_OP		: BOOL;

	Status_Log		: BYTE;
	Status_Vis 		: DWORD;
END_VAR
VAR
	Curve		: CHARCURVE;
	Curve_Err	: BYTE;

	Ctrl_Out_Time	:	REAL;
	PwmTmr			:   TON := (PT:=T#5s);

	fClose		: BOOL;	(* Valve is completly closed *)
	fOpen		: BOOL;	(* Valve is completely open  *)
	CloseCtr	: BYTE;	(* Close counter *)
	OpenCtr		: BYTE; (* Open counter  *)

	aTemp		: ARRAY [1..20] OF INT;
	meanTemp	: INT;
	sum			: INT := 0;
	Tmr			: TON := (PT:=T#1s);
	index		: BYTE;
	i			: BYTE;
	fCtrl_Err	: BOOL;		(* TRUE: Ctrl_Err>0, FALSE: Ctrl_Err<0 *)
END_VAR



VAR_INPUT RETAIN
	Local_VRD_TAlarm: INT;

	Ctrl_ErrGate	: INT:=5;		(* Error gate - 0.5°C *)
	Ctrl_Kp			: REAL:=1;(*5;*)		(* Proportional factor *)
	Ctrl_Kd			: REAL:=5;(*10;*)  	(* Derivative factor *)
	Chk_ErrGate		: INT:=1000; 		(* Check error gate *)



END_VAR
(* Check initialization *)
IF NOT InitOK THEN Init(); END_IF

(* Check max temperature *)
IF TEMP>Plant_VRD_TAlarm THEN
	IF NOT Alarm1 THEN
		Alarm1:=TRUE;
		LogEv(EL_AlarmStop,EO_VRD,ID,3,'VRD_Overtemperature');
	END_IF
END_IF

(* Check climatic setup *)
IF NOT CLIM.InitOK THEN	DefaultClim(); END_IF;
(* Calculate Setpoint *)
Curve(	IN:= T_AMB,	N:= 5, P:= CLIM.Points,			(* Given the x value as input, the corresponding y value as output is returned, if it matches the crve designed by array of points *)
		OUT=> Ctrl_SetPointNew, ERR=> Curve_Err );
IF Curve_Err>0 OR Ctrl_SetPoint>Plant_VRD_TMax THEN
	IF Ctrl_SetPoint>Plant_VRD_TMax THEN
		Ctrl_SetPoint:=Plant_VRD_TMax;
	ELSE
		Ctrl_SetPoint:=Plant_VRD_TDefault;
	END_IF
	IF NOT Warning THEN
		Warning:=TRUE;
		LogEv(EL_Wrn,EO_VRD,ID,2,'VRD_Climatic_Error');
	END_IF
ELSE
	Delta_SetPoint := ABS(Ctrl_SetPoint - Ctrl_SetPointNew);
	IF Delta_SetPoint>Ctrl_SetPointGate THEN Ctrl_SetPoint := Ctrl_SetPointNew; END_IF

	Warning:=FALSE;
END_IF

Ctrl_SetPoint:=Ctrl_SetPoint+OffsetBoost;

(* Execute control loop [T=500ms] *)
IF RUN AND (NOT Alarm1) THEN
	(* Calculate error *)
	Ctrl_Err:=Ctrl_SetPoint-TEMP;
	(* Init/restart operations *)
	IF NOT Ctrl_Init THEN
		Ctrl_Accel:=0;
		Ctrl_AccelTmr:=0;
		Ctrl_Err0:=Ctrl_Err;
		Ctrl_Out:=0;
		Ctrl_Init:=TRUE;
	END_IF
	(* Calculate acceleration *)
	IF ABS(Ctrl_Err-Ctrl_Err0)>Ctrl_AccelGate OR Ctrl_AccelTmr>2 THEN
		Ctrl_Accel:=INT_TO_REAL(Ctrl_Err-Ctrl_Err0)/WORD_TO_REAL(1+Ctrl_AccelTmr);
		Ctrl_AccelTmr:=0;
		Ctrl_Err0:=Ctrl_Err;
	ELSE
		Ctrl_AccelTmr:=Ctrl_AccelTmr+1;
	END_IF

	(* Gate error *)
	IF ABS(Ctrl_Err)>Ctrl_ErrGate THEN
		(* Control loop *)
		Ctrl_Out:=Ctrl_Out+(Ctrl_Kp*Ctrl_Err)+(Ctrl_Kd*Ctrl_Accel);

		(* Limiter and Output *)
		Ctrl_Out_Time := LIMIT(0,ABS(Ctrl_Out),TIME_TO_REAL(Tpwm));

		PwmTmr(IN:=NOT PwmTmr.Q);

		IF PwmTmr.ET>=REAL_TO_TIME(Ctrl_Out_Time) THEN
			(* Stop corretction *)
			OUT_OP := FALSE;
			OUT_CL := FALSE;
		END_IF

		IF PwmTmr.Q THEN
			(* Adjust valve position *)
			IF fFeedback THEN
				IF Ctrl_Err>0 AND NOT fOpen THEN OUT_OP := TRUE; END_IF		(* If valve yet open don't drive physical output *)
				IF Ctrl_Err<0 AND NOT fClose THEN OUT_CL := TRUE; END_IF	(* If valve yet close don't drive physical output *)
			ELSE
				IF Ctrl_Err>0 THEN OUT_OP := TRUE; END_IF
				IF Ctrl_Err<0 THEN OUT_CL := TRUE; END_IF
			END_IF

			PwmTmr.PT := Tpwm;
		END_IF
	END_IF
ELSE
	OUT_CL := TRUE; (* forzatura serranda in chiusura se il circolatore corrispettivo non è comandato *)
	Ctrl_Init:=FALSE;
END_IF

(* If there is an hardware feedback (such as 0-10V, potentiometer, ...) check it otherwise try to rebuild it *)
IF fFeedback THEN CheckFeedback();
ELSE BuildFeedback();
END_IF


(* Status color *)
   IF Alarm1 THEN Status_Log:=2; Status_Vis:=COLOR_RED;
ELSIF Warning  OR Alarm2 THEN Status_Log:=1; Status_Vis:=COLOR_YELLOW;
                       ELSE Status_Log:=0; Status_Vis:=SEL(RUN,COLOR_LIGHT_GREEN,COLOR_GREEN);
END_IF
END_FUNCTION_BLOCK
ACTION AddLogData:
Logger.s1:=INSERT('&VRD=',BYTE_TO_STRING(ID),4);
IF ID<10 THEN Logger.s1:=INSERT(Logger.s1,'0',4); END_IF

Logger.s1:=CONCAT(Logger.s1,INT_TO_STRING(Ctrl_SetPoint));				Logger.s1:=CONCAT(Logger.s1,';');
Logger.s1:=CONCAT(Logger.s1,'0');	(* Bypass *)						Logger.s1:=CONCAT(Logger.s1,';');

IF fFeedback THEN Logger.s1:=CONCAT(Logger.s1,WORD_TO_STRING(STATUS));
ELSE Logger.s1:=CONCAT(Logger.s1,'0');	(* Bypass *)
END_IF

Logger.s1:=CONCAT(Logger.s1,';');
Logger.s1:=CONCAT(Logger.s1,WORD_TO_STRING(Status_Log));

Logger.s1:=CONCAT(Logger.s1,';');
Logger.s1:=CONCAT(Logger.s1,SEL(OUT_OP,'0','100'));
Logger.s1:=CONCAT(Logger.s1,';');
Logger.s1:=CONCAT(Logger.s1,SEL(OUT_CL,'0','100'));




ADDSTRING(ADR(Logger.TData), ADR(Logger.s1), Logger.TLen);
END_ACTION
ACTION BuildFeedback:
(* Comparison is taken between actual temperature vs windowed mean value OF last 20 temperature
   (check is carried out every second)	*)
IF RUN AND (NOT Alarm1) THEN

	IF Ctrl_Err>0 THEN
		IF NOT fCtrl_Err THEN index := 0; END_IF
		fCtrl_Err := TRUE;
	ELSE
		IF fCtrl_Err THEN index := 0; END_IF
		fCtrl_Err := FALSE;
	END_IF

	(* Temperature is lower than setpoint -->> Should increase *)
	Tmr(IN:=NOT Tmr.Q);

	IF Tmr.Q THEN

		IF index<21 THEN
			(* Fullfil temperature array *)
			aTemp[index] := TEMP;
			index := index + 1;

			IF index=20 THEN
				FOR i:=1 TO 20 BY 1 DO sum := sum + aTemp[i]; END_FOR
			END_IF
		ELSE
			(* Calculate mean value *)
			meanTemp := sum/20;

			IF (fCtrl_Err AND TEMP<meanTemp) OR (NOT fCtrl_Err AND TEMP>meanTemp) THEN

				IF Chk_Cnt>Chk_CntSecAlarm THEN
					IF NOT Alarm2 THEN
						Alarm2:=TRUE;
						LogEv(EL_wrn,EO_VRD,ID,2,'VRD_Position_Error');
					END_IF
				ELSE
					Chk_Cnt := Chk_Cnt+1;
				END_IF

			ELSE
				(* Reset counter and alarm flag *)
				Chk_Cnt:=0;
				Alarm2:=FALSE;
			END_IF

			sum := 0;	(* Reset sum counter *)

			(* Shift array removing oldest value *)
			FOR i:=1 TO 20 BY 1 DO
				aTemp[i-1] := aTemp[i];
				sum := sum + aTemp[i];
			END_FOR

			aTemp[20] := TEMP;			(* Last temperature value is new one *)
			sum := sum + aTemp[20];		(* Update sum *)
		END_IF
	END_IF
END_IF
END_ACTION
ACTION CheckFeedback:
(* Check position *)
IF Status=ValveCloseRes THEN

	CloseCtr := CloseCtr+1;
	IF CloseCtr=ValvePosCheck THEN	fClose := TRUE;	END_IF

ELSIF Status=ValveOpenRes THEN

	OpenCtr := OpenCtr+1;
	IF OpenCtr=ValvePosCheck THEN	fOpen := TRUE;	END_IF

ELSE

	fClose := FALSE;
	fOpen  := FALSE;

END_IF

(* Check position error *)


(* 0xEC00 corresponds to 0ohm, while other values are linear from 20 (10ohm -> 1%) to 2000 (1Kohm -> 100%) *)
IF Status = 16#EC00 THEN Chk_Err := Ctrl_Out;
ELSE
   Chk_Err := Ctrl_Out - Status/2;
END_IF

IF ( Chk_Err<-Chk_ErrGate OR Chk_Err>Chk_ErrGate ) THEN
	IF Chk_Cnt>Chk_CntAlarm THEN
		IF NOT Alarm2 THEN
			Alarm2:=TRUE;
			LogEv(EL_wrn,EO_VRD,ID,2,'VRD_Position_Error');
		END_IF
	ELSE
		Chk_Cnt:=Chk_Cnt+1;
	END_IF
ELSE
	Chk_Cnt:=0;
	Alarm2:=FALSE;
END_IF
END_ACTION
ACTION DefaultClim:
IF CLIM.Points[0].X=0 THEN
CLIM.Points[0].X:=-300; CLIM.Points[0].Y:=850;
CLIM.Points[1].X:=-70;  CLIM.Points[1].Y:=750;
CLIM.Points[2].X:= 100; CLIM.Points[2].Y:=630;
CLIM.Points[3].X:= 200; CLIM.Points[3].Y:=250;
CLIM.Points[4].X:= 500; CLIM.Points[4].Y:=200;
END_IF
CLIM.InitOK:=TRUE;
LogEv(EL_Wrn,EO_VRD,ID,1,'Climatic_Default');
END_ACTION
ACTION Init:
(* End initialization *)
InitOK:=TRUE;
END_ACTION

(* POU Plant_Objects/obj_ZTHL, ST *)
FUNCTION_BLOCK obj_ZTHL
(* === ZIGBEE AMBIENT SENSORS MT-200 ===
   v1.0[07/05/05] - Create
*)
VAR CONSTANT
	(* States *)
	WAIT_STATE			:	BYTE := 0;
	STATUS_REQUEST		:	BYTE := 1;
	LQI_REQUEST			:	BYTE := 2;
	MEAS_REQUEST		:	BYTE := 3;
	END_READ			:	BYTE := 4;
	ERROR_STATE			:	BYTE := 100;

	LQI_Threshold		:	WORD := 100;		(* Zigbee link quality minimum value *)
	LowBattVoltage		:	WORD := 270;		(* Battery is considered low when reaches 1.35V each *)
END_VAR
VAR_INPUT
	(* Settings *)
	ID				: BYTE;
	Address			: BYTE;

	Refresh_Period	: TIME:=t#5m;
	(* Controls *)
	Refresh_Auto	: BOOL:=TRUE; (* Enable automatic refresh *)
	Refresh_Now		: BOOL; 	  (* Force an immediate refresh *)

	(* Limits *)
	Tmin			: INT := 50;
	Tmax			: INT := 400;
END_VAR
VAR_IN_OUT
	(* Interface *)
	MODBUS			: obj_MODBUS_TCP;
END_VAR
VAR_OUTPUT
	OUT_STATUS		: WORD;
	OUT_TEMP		: INT;	(* Temperatura misurata [°C/10] *)
	OUT_HYGRO		: INT;	(* Umidità misurata [%] *)
	OUT_LUX			: INT;	(* Luce misurata [lux] *)
	OUT_VBATT		: INT;	(* Tensione misurata dalla batteria [V/100] *)

	OUT_LQI			: BYTE;

	ERR				: BOOL;

	(* Status *)
	Status_Log		: BYTE;
	Status_Vis 		: DWORD;
END_VAR
VAR
	dly 	 		: TON := (PT:=t#5s);

	sta				: BYTE;
	retry	 		: BYTE;

	Status			: FLT_EVENT;
	Quality			: FLT_EVENT;
	NoSignal		: FLT_EVENT;
	Battery			: FLT_EVENT;
	Temperature		: FLT_EVENT := (INITEV:=FALSE);
	Alarm			: FLT_EVENT;

	AlarmCtr		: BYTE;
	WarningCtr		: BYTE;

END_VAR
CASE sta OF
	WAIT_STATE: (* === Wait update signals *)
		dly(IN:=NOT (dly.Q OR Refresh_Now OR (NOT Refresh_Auto)));
		IF dly.Q OR Refresh_Now THEN
			dly.PT:=Refresh_Period;
			Refresh_Now:=FALSE;
			sta:=STATUS_REQUEST;
		(*	sta:=LQI_REQUEST; *)
		END_IF

	STATUS_REQUEST:	(* Node status *)
		IF NOT (MODBUS.MB_Lock OR MODBUS.MB_Start) THEN
			MODBUS.MB_Lock:=TRUE;
			MODBUS.ID:=ID;
			MODBUS.MB_MASTER.bUNIT_ID := Address;
			MODBUS.MB_MASTER.bFUNCTION_CODE:=16#03;
			MODBUS.MB_MASTER.wREAD_ADDRESS:=16#0D;
			MODBUS.MB_MASTER.wREAD_QUANTITY:=16#1;
			MODBUS.MB_Start:=TRUE;
			sta:=LQI_REQUEST;
		END_IF

	LQI_REQUEST:	(* Link quality *)
		IF NOT MODBUS.MB_Start THEN
			IF MODBUS.MB_MASTER.wERROR<>MB_NO_ERROR THEN
				sta:=ERROR_STATE;
			ELSE
				OUT_STATUS	:=	MODBUS.MB_READBUF[0];

				MODBUS.ID:=ID;
				MODBUS.MB_MASTER.bUNIT_ID := Address;
				MODBUS.MB_MASTER.bFUNCTION_CODE:=16#03;
				MODBUS.MB_MASTER.wREAD_ADDRESS:=16#01;
				MODBUS.MB_MASTER.wREAD_QUANTITY:=16#1;
				MODBUS.MB_Start:=TRUE;

				sta:=MEAS_REQUEST;
			END_IF
		END_IF

	MEAS_REQUEST:	(* Measurements *)
		IF NOT MODBUS.MB_Start THEN
			IF MODBUS.MB_MASTER.wERROR<>MB_NO_ERROR THEN
				sta:=ERROR_STATE;
			ELSE

				OUT_LQI	:=	WORD_TO_BYTE(MODBUS.MB_READBUF[0]);

				MODBUS.ID:=ID;
				MODBUS.MB_MASTER.bUNIT_ID := Address;
				MODBUS.MB_MASTER.bFUNCTION_CODE:=16#03;
				MODBUS.MB_MASTER.wREAD_ADDRESS:=16#14;
				MODBUS.MB_MASTER.wREAD_QUANTITY:=16#5;
				MODBUS.MB_Start:=TRUE;

				sta:=END_READ;
			END_IF
		END_IF

	END_READ:	IF NOT MODBUS.MB_Start THEN
			IF MODBUS.MB_MASTER.wERROR<>MB_NO_ERROR THEN
				sta:=ERROR_STATE;
			ELSE
				OUT_TEMP	:=	WORD_TO_INT(MODBUS.MB_READBUF[0]);
				OUT_HYGRO	:=	WORD_TO_INT(MODBUS.MB_READBUF[1]);
				OUT_LUX		:=	WORD_TO_INT(MODBUS.MB_READBUF[2]);
				OUT_VBATT	:=	WORD_TO_INT(MODBUS.MB_READBUF[3]);
				sta:=WAIT_STATE;
				MODBUS.MB_Lock:=FALSE;
			END_IF
		END_IF

	ERROR_STATE:
			MODBUS.MB_Lock:=FALSE;
			(* Retries *)
			retry:=retry+1;
			IF retry>3 THEN
				retry:=0;
				IF Status_Log<>2 THEN
					LogEv(EL_Alarm,EO_ZTHL,ID,4,'');
				END_IF
				Status_Log:=2;
				Status_Vis:=COLOR_RED;
			END_IF
			sta:=WAIT_STATE;

ELSE
			sta:=WAIT_STATE;
END_CASE

(* Check Status *)
Status(IN:=(OUT_STATUS<>1));

IF Status.EVH THEN LogEv(EL_Alarm,EO_ZTHL,ID,3,'NodoZTHL_OffLine'); END_IF

(* Check if there is signal (Link Quality different from 0) *)
NoSignal(IN:=(OUT_LQI=0));

IF NoSignal.EVH THEN
	LogEv(EL_Alarm,EO_ZTHL,ID,7,'');
	AlarmCtr := AlarmCtr + 1;
END_IF

IF NoSignal.EVL THEN AlarmCtr := SEL(AlarmCtr=0,AlarmCtr-1,0); END_IF

(* Check Link Quality *)
Quality(IN:=(OUT_LQI < LQI_Threshold));

IF Quality.EVL THEN
	LogEv(EL_Wrn,EO_ZTHL,ID,2,WORD_TO_STRING(OUT_LQI));
	WarningCtr := WarningCtr + 1;
END_IF

IF Quality.EVH THEN WarningCtr := SEL(WarningCtr=0,WarningCtr-1,0); END_IF

(* If probe (node) is present proceed checking other warnings, otherwise don't transmit anything *)
IF OUT_LQI>0 THEN (* AND OUT_STATUS=1 THEN *)

	(* Check battery voltage *)
	Battery(IN:=(OUT_VBATT<LowBattVoltage));

	IF Battery.EVH THEN
		LogEv(EL_Wrn,EO_ZTHL,ID,6,'');
		WarningCtr := WarningCtr + 1;
	END_IF

	IF Battery.EVL THEN WarningCtr := SEL(WarningCtr=0,WarningCtr-1,0); END_IF

	(* Check Node temperature *)
	Temperature(IN:=(OUT_TEMP<Tmin OR OUT_TEMP>Tmax));

	IF Temperature.EVH THEN
		LogEv(EL_Wrn,EO_ZTHL,ID,5,INT_TO_STRING(OUT_TEMP));
		WarningCtr := WarningCtr + 1;
	END_IF

	IF Temperature.EVL THEN WarningCtr := SEL(WarningCtr=0,WarningCtr-1,0); END_IF

ELSE
	OUT_TEMP 	:= 0;
	OUT_HYGRO 	:= 0;
	OUT_LUX 	:= 0;
	OUT_VBATT 	:= 0;
END_IF

Alarm(IN:=(AlarmCtr=0 AND WarningCtr=0));

IF Alarm.EVH THEN LogEv(EL_Log,EO_ZTHL,ID,1,'Sonda_Ambiente_Errore'); END_IF

IF AlarmCtr>0 OR (OUT_STATUS<>1) THEN
	Status_Log := 2;
	Status_Vis := COLOR_RED;
	ERR := TRUE;
ELSIF WarningCtr>0 THEN
	Status_Log := 1;
	Status_Vis := COLOR_YELLOW;
	ERR := FALSE;
ELSE
	Status_Log := 0;
	Status_Vis := COLOR_GREEN;
	ERR := FALSE;
END_IF
END_FUNCTION_BLOCK
ACTION AddLogData:
Logger.s1:=INSERT('&ZTHL=',BYTE_TO_STRING(ID),5);
IF ID<10 THEN Logger.s1:=INSERT(Logger.s1,'0',5); END_IF

Logger.s1:=CONCAT(Logger.s1,BYTE_TO_STRING(OUT_LQI));			Logger.s1:=CONCAT(Logger.s1,';');
Logger.s1:=CONCAT(Logger.s1,INT_TO_STRING(OUT_TEMP ));			Logger.s1:=CONCAT(Logger.s1,';');
Logger.s1:=CONCAT(Logger.s1,INT_TO_STRING(OUT_HYGRO ));			Logger.s1:=CONCAT(Logger.s1,';');
Logger.s1:=CONCAT(Logger.s1,INT_TO_STRING(OUT_LUX));			Logger.s1:=CONCAT(Logger.s1,';');
Logger.s1:=CONCAT(Logger.s1,INT_TO_STRING(OUT_VBATT));			Logger.s1:=CONCAT(Logger.s1,';');

Logger.s1:=CONCAT(Logger.s1,BYTE_TO_STRING(Status_Log));
ADDSTRING(ADR(Logger.TData), ADR(Logger.s1), Logger.TLen);
END_ACTION

(* POU Utils Functions/PLANT_STATUS, ST *)
FUNCTION_BLOCK PLANT_STATUS
VAR_INPUT
	obj_Status		:	WORD;
END_VAR
VAR_OUTPUT
END_VAR
VAR
	PLANT_STATUS	:	WORD;

	Pwm				:	TON := (PT:=T#1s);
END_VAR
CASE plant_Status OF

	0:	(* Plant OK - Everything works well *)
		(*Pwm(IN:=FALSE);	*)						(* Stop timer if running *)
		LAMP_AL := FALSE;						(* Keep the lamp switched off *)

	(*1:	(* Plant in warning *)
		Pwm(IN:= NOT(Pwm.Q));

		IF Pwm.Q THEN
			LAMP_AL := NOT LAMP_AL;				(* Toggle output *)
		END_IF*)

	2:	(* Plant in alarm *)
		(*Pwm(IN:=FALSE);	*)						(* Stop timer if running *)
		LAMP_AL	:= TRUE;						(* Keep the lamp switched on *)

END_CASE

plant_Status := 0;		(* Reset plant status *)
END_FUNCTION_BLOCK
ACTION UpdateStatus:
IF plant_Status = 2 THEN

	RETURN;					(* If plant already in alarm condition do nothing *)

ELSE

		IF obj_Status <> 0 THEN
			plant_Status := obj_Status;			(* If plant in warning/normal condition and current object in alarm, update plant status *)
		END_IF
END_IF
END_ACTION

(* POU PLC_WDT, ST *)
FUNCTION PLC_WDT: DWORD VAR_INPUT dwEvent: DWORD; dwFilter: DWORD; dwOwner: DWORD; END_VAR
LogEv(EL_AlarmStop,EO_SYS,1,10,'Watchdog');
END_FUNCTION

(* POU Utils Functions/RAW16TOHEXSTR, ST *)
FUNCTION RAW16TOHEXSTR : STRING(128)
VAR_INPUT
	pData: POINTER TO BYTE;
	DataLen: BYTE;
END_VAR
VAR
	pt: POINTER TO BYTE;
	xl: BYTE;
END_VAR
pt:=ADR(RAW16TOHEXSTR);
xl:=0;

WHILE DataLen>0 AND xl<120 DO

	pData:=pData+1;

	pt^ := (pData^ / 16#10) + 48 + (((pData^ / 16#10)/10)*7);
	pt:=pt+1;
	pt^ := (pData^ AND 16#0F)  + 48 + (((pData^ AND 16#0F)/10)*7);
	pt:=pt+1;

	pData:=pData-1;

	pt^ := (pData^ / 16#10) + 48 + (((pData^ / 16#10)/10)*7);
	pt:=pt+1;
	pt^ := (pData^ AND 16#0F)  + 48 + (((pData^ AND 16#0F)/10)*7);
	pt:=pt+1;

	xl:=xl+4;

	DataLen:=DataLen-2;
	pData:=pData+2;

END_WHILE

pt^:=0;
END_FUNCTION

(* POU Utils/RTC_Update, ST *)
FUNCTION RTC_Update : BOOL
VAR
	T: DT;
	TS: STRING;
	TS2: STRING;
	Hour: BYTE;
	Minute: BYTE;
END_VAR
(* Get RTC time *)
T:=SysRtcGetTime(TRUE);
Sys.Time_CT_DT:=T;
(* Calculate variables *)
TS:=DT_TO_STRING(T);
Sys.Time_LogString:=DELETE(STR:=TS, LEN:=3, POS:=1);
TS2:=MID(STR:=TS, LEN:=4, POS:= 4); Sys.Time_Year 	:=STRING_TO_WORD(TS2);
TS2:=MID(STR:=TS, LEN:=2, POS:= 9); Sys.Time_Month	:=STRING_TO_BYTE(TS2);
TS2:=MID(STR:=TS, LEN:=2, POS:=12); Sys.Time_Day  	:=STRING_TO_BYTE(TS2);
Sys.Time_CT_Day:=(32*(Sys.Time_Month-1)+Sys.Time_Day-1);
TS2:=MID(STR:=TS, LEN:=2, POS:=15); Hour			:=STRING_TO_BYTE(TS2);
TS2:=MID(STR:=TS, LEN:=2, POS:=18); Minute		 	:=STRING_TO_BYTE(TS2);
Sys.Time_Hour := Hour;
Sys.Time_Minute := Minute;
Sys.Time_CT_Quarter:=Hour*4+(Minute/15);
END_FUNCTION

(* POU Utils Functions/SHIFT_ARRAY, ST *)
FUNCTION SHIFT_ARRAY : BOOL
VAR_INPUT
	pData	:	POINTER TO ARRAY [1..2] OF WORD;
	Size	:	BYTE;
END_VAR
VAR
	pNew	:	POINTER TO WORD;
	i		:	BYTE;
END_VAR
(* Shift right *)
FOR i:=1 TO (Size-1) BY 1 DO

	(*pNew := pData + 1;*)
	pData^[i] := pData^[i+1];
	(*pData := pData + 1;*)

END_FOR
END_FUNCTION

(* Visualisation PLC_VISU
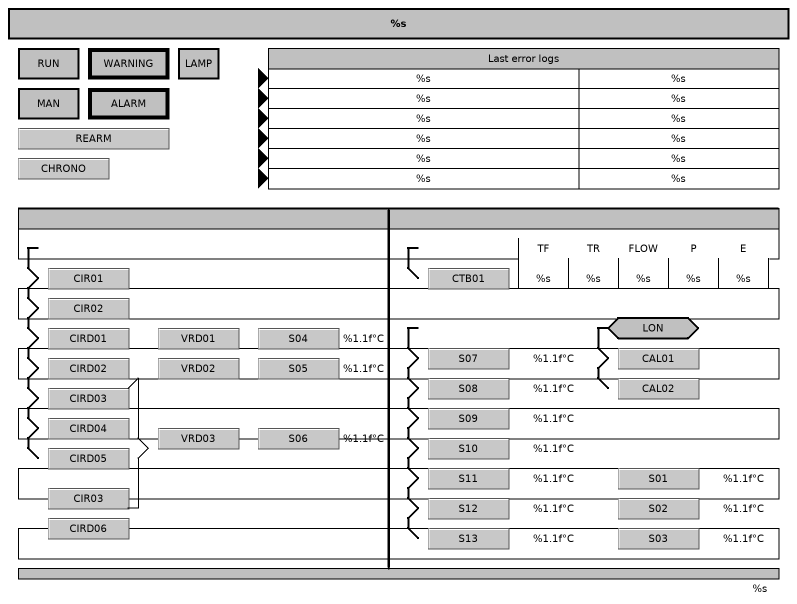
rectangle at (10,10)-(791,41): text "%s"; shows .Plant_NAME
rectangle at (530,580)-(771,601): text "%s"; shows Sys.Time_LogString
rounded rectangle at (20,50)-(81,81): text "RUN"; alarm colour if NOT Mode_Manual; runs INTERN ASSIGN Mode_Manual:=(FALSE)
rounded rectangle at (20,90)-(81,121): text "MAN"; alarm colour if Mode_Manual; runs INTERN ASSIGN Mode_Manual:=(TRUE)
rectangle at (580,70)-(781,91): text "%s"; shows Sys.LastLogs_Msg[0]
polygon at (260,170)-(270,190): invisible if Sys.LastLogs_Idx<>0
rectangle at (580,90)-(781,111): text "%s"; shows Sys.LastLogs_Msg[1]
polygon at (260,70)-(270,90): invisible if Sys.LastLogs_Idx<>1
rectangle at (580,110)-(781,131): text "%s"; shows Sys.LastLogs_Msg[2]
polygon at (260,90)-(270,110): invisible if Sys.LastLogs_Idx<>2
rectangle at (580,130)-(781,151): text "%s"; shows Sys.LastLogs_Msg[3]
polygon at (260,110)-(270,130): invisible if Sys.LastLogs_Idx<>3
rectangle at (580,150)-(781,171): text "%s"; shows Sys.LastLogs_Msg[4]
polygon at (260,130)-(270,150): invisible if Sys.LastLogs_Idx<>4
rectangle at (580,170)-(781,191): text "%s"; shows Sys.LastLogs_Msg[5]
polygon at (260,150)-(270,170): invisible if Sys.LastLogs_Idx<>5
rectangle at (270,70)-(581,91): text "%s"; shows Sys.LastLogs_Dat[0]
rectangle at (270,90)-(581,111): text "%s"; shows Sys.LastLogs_Dat[1]
rectangle at (270,110)-(581,131): text "%s"; shows Sys.LastLogs_Dat[2]
rectangle at (270,130)-(581,151): text "%s"; shows Sys.LastLogs_Dat[3]
rectangle at (270,150)-(581,171): text "%s"; shows Sys.LastLogs_Dat[4]
rectangle at (270,170)-(581,191): text "%s"; shows Sys.LastLogs_Dat[5]
rectangle at (90,90)-(171,121): text "ALARM"; alarm colour if Sys.Alarm; runs INTERN ASSIGN Mode_Manual:=(FALSE)
rectangle at (90,50)-(171,81): text "WARNING"; alarm colour if Sys.Warning; runs INTERN ASSIGN Mode_Manual:=(TRUE)
button at (20,130)-(171,151): text "REARM"; runs INTERN ASSIGN Sys.Alarm:=(FALSE);INTERN ASSIGN Sys.Warning:=(FALSE)
button at (430,270)-(511,291): text "CTB01"
rectangle at (270,50)-(781,71): text "Last error logs"
rectangle at (520,240)-(571,261): text "TF"
rectangle at (620,240)-(671,261): text "FLOW"
rectangle at (670,240)-(721,261): text "P"
rectangle at (720,240)-(771,261): text "E"
rectangle at (570,240)-(621,261): text "TR"
rectangle at (520,270)-(571,291): text "%s"; shows .CTB01.M1.utFTemp.Value
rectangle at (620,270)-(671,291): text "%s"; shows .CTB01.M1.utFlow.Value
rectangle at (670,270)-(721,291): text "%s"; shows CTB01.M1.utPower.Value
rectangle at (720,270)-(771,291): text "%s"; shows CTB01.M1.utEnergy.Value
rectangle at (570,270)-(621,291): text "%s"; shows .CTB01.M1.utRTemp.Value
button at (50,330)-(131,351): text "CIRD01"
button at (50,360)-(131,381): text "CIRD02"
button at (50,390)-(131,411): text "CIRD03"
button at (50,270)-(131,291): text "CIR01"
button at (50,420)-(131,441): text "CIRD04"
button at (50,300)-(131,321): text "CIR02"
button at (620,470)-(701,491): text "S01"; opens Vis_VRD02
button at (620,500)-(701,521): text "S02"; opens Vis_VRD02
button at (620,530)-(701,551): text "S03"; opens Vis_VRD02
button at (430,350)-(511,371): text "S07"; opens Vis_VRD02
button at (430,380)-(511,401): text "S08"; opens Vis_VRD02
button at (430,410)-(511,431): text "S09"; opens Vis_VRD02
button at (430,440)-(511,461): text "S10"; opens Vis_VRD02
button at (430,470)-(511,491): text "S11"; opens Vis_VRD02
button at (430,500)-(511,521): text "S12"; opens Vis_VRD02
button at (430,530)-(511,551): text "S13"; opens Vis_VRD02
rectangle at (700,470)-(791,491): text "%1.1f°C"; shows INT_TO_REAL(.TPV01.IN)/10
rectangle at (700,500)-(791,521): text "%1.1f°C"; shows INT_TO_REAL(.TPV02.IN)/10
rectangle at (700,530)-(791,551): text "%1.1f°C"; shows INT_TO_REAL(.TPV03.IN)/10
rectangle at (510,350)-(601,371): text "%1.1f°C"; shows INT_TO_REAL(ZTHL07.OUT_TEMP)/10
rectangle at (510,380)-(601,401): text "%1.1f°C"; shows INT_TO_REAL(ZTHL08.OUT_TEMP)/10
rectangle at (510,410)-(601,431): text "%1.1f°C"; shows INT_TO_REAL(.ZTHL09.OUT_TEMP)/10
rectangle at (510,440)-(601,461): text "%1.1f°C"; shows INT_TO_REAL(ZTHL10.OUT_TEMP)/10
rectangle at (510,470)-(601,491): text "%1.1f°C"; shows INT_TO_REAL(ZTHL11.OUT_TEMP)/10
rectangle at (510,500)-(601,521): text "%1.1f°C"; shows INT_TO_REAL(ZTHL12.OUT_TEMP)/10
rectangle at (510,530)-(601,551): text "%1.1f°C"; shows INT_TO_REAL(ZTHL13.OUT_TEMP)/10
button at (620,350)-(701,371): text "CAL01"; opens Vis_CAL01
polygon at (610,320)-(700,340): text "LON"
button at (620,380)-(701,401): text "CAL02"; opens Vis_CAL01
button at (50,450)-(131,471): text "CIRD05"
button at (50,520)-(131,541): text "CIRD06"
button at (160,330)-(241,351): text "VRD01"; opens Vis_VRD02
button at (160,360)-(241,381): text "VRD02"; opens Vis_VRD02
rounded rectangle at (180,50)-(221,81): text "LAMP"; alarm colour if LAMP_AL
button at (160,430)-(241,451): text "VRD03"; opens Vis_VRD02
button at (50,490)-(131,511): text "CIR03"
button at (260,330)-(341,351): text "S04"; opens Vis_VRD02
button at (260,360)-(341,381): text "S05"; opens Vis_VRD02
button at (260,430)-(341,451): text "S06"; opens Vis_VRD02
rectangle at (340,330)-(391,351): text "%1.1f°C"; shows INT_TO_REAL(TPV04.IN)/10
rectangle at (340,360)-(391,381): text "%1.1f°C"; shows INT_TO_REAL(.TPV05.IN)/10
rectangle at (340,430)-(391,451): text "%1.1f°C"; shows INT_TO_REAL(.TPV06.IN)/10
button at (20,160)-(111,181): text "CHRONO"; opens VIS_CHONOEDITOR
34 more shapes without text or variables
31 elements of other kinds (tables, trends, ...) not read
*)

(* Visualisation VIS_CAL01
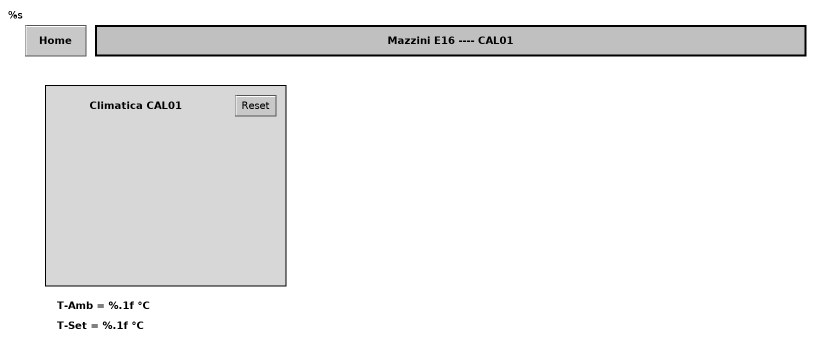
rectangle at (40,300)-(181,321): text "T-Set = %.1f °C"; shows INT_TO_REAL(CAL01.CFD_SetPoint.iSnvtTempP)/100
rectangle at (0,0)-(0,0): text "%s"; shows CAL01_Clima.Points[INDEX].X; invisible if INDEX>4; editable
rectangle at (0,0)-(0,0): text "%s"; shows CAL01_Clima.Points[INDEX].Y; invisible if INDEX>4; editable
rectangle at (40,280)-(181,301): text "T-Amb = %.1f °C"; shows INT_TO_REAL(.T_AMB)/10; alarm colour if T_AMB>2000
rectangle at (40,80)-(201,101): text "Climatica CAL01"
button at (220,80)-(261,101): text "Reset"; runs INTERN ASSIGN CAL01_Clima.InitOK:=(FALSE)
rectangle at (80,10)-(791,41): text "Mazzini E16 ---- CAL01"
button at (10,10)-(71,41): text "Home"; opens PLC_VISU
1 more shapes without text or variables
*)

(* Visualisation VIS_CAL02
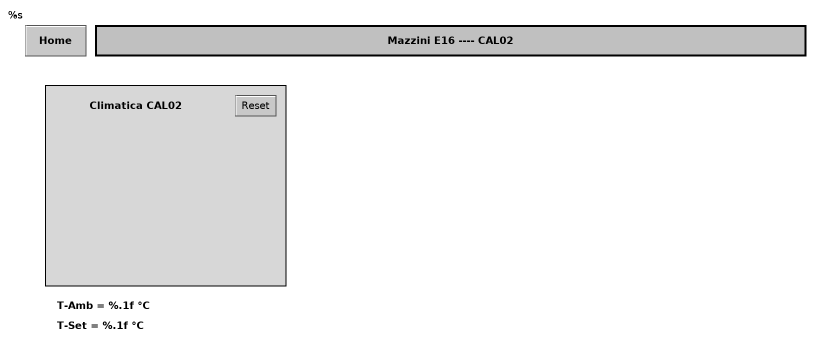
rectangle at (40,300)-(181,321): text "T-Set = %.1f °C"; shows INT_TO_REAL(CAL02.CFD_SetPoint.iSnvtTempP)/100
rectangle at (0,0)-(0,0): text "%s"; shows CAL01_Clima.Points[INDEX].X; invisible if INDEX>4; editable
rectangle at (0,0)-(0,0): text "%s"; shows CAL01_Clima.Points[INDEX].Y; invisible if INDEX>4; editable
rectangle at (40,280)-(181,301): text "T-Amb = %.1f °C"; shows INT_TO_REAL(.T_AMB)/10; alarm colour if T_AMB>2000
rectangle at (40,80)-(201,101): text "Climatica CAL02"
button at (220,80)-(261,101): text "Reset"; runs INTERN ASSIGN CAL01_Clima.InitOK:=(FALSE)
rectangle at (80,10)-(791,41): text "Mazzini E16 ---- CAL02"
button at (10,10)-(71,41): text "Home"; opens PLC_VISU
1 more shapes without text or variables
*)

(* Visualisation VIS_CHONOEDITOR
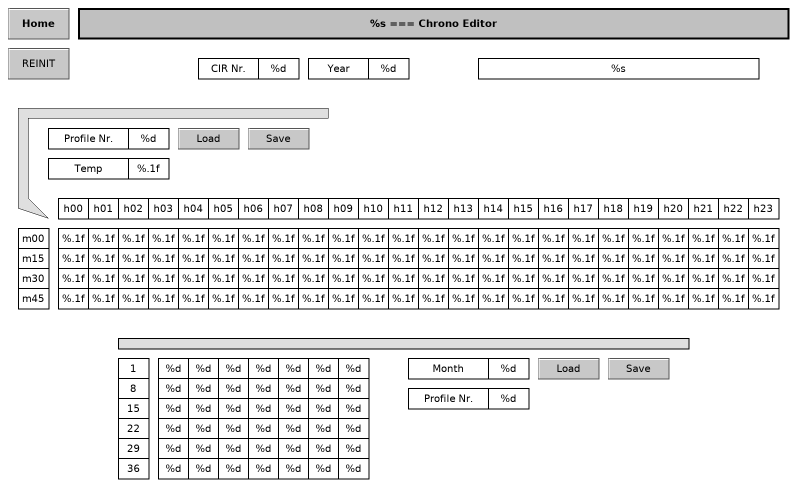
rectangle at (200,60)-(261,81): text "CIR Nr."
rectangle at (260,60)-(301,81): text "%d"; shows CronEd.CN_Sel; alarm colour if CronEd.CN_Sel<>CronEd.CN_Act; editable 1..250
rectangle at (50,130)-(131,151): text "Profile Nr."
rectangle at (130,130)-(171,151): text "%d"; shows CronEd.PR_Sel; alarm colour if CronEd.PR_Sel<>CronEd.PR_Act; editable 1..10
rectangle at (50,160)-(131,181): text "Temp"
rectangle at (130,160)-(171,181): text "%.1f"; shows CronEd.PR_TT; editable
button at (180,130)-(241,151): text "Load"; toggles CronEd.PR_Load
button at (250,130)-(311,151): text "Save"; toggles CronEd.PR_Save
rectangle at (20,230)-(51,251): text "m00"
rectangle at (20,250)-(51,271): text "m15"
rectangle at (20,270)-(51,291): text "m30"
rectangle at (20,290)-(51,311): text "m45"
rectangle at (80,10)-(791,41): text "%s === Chrono Editor"; shows .Plant_NAME
button at (10,10)-(71,41): text "Home"; opens PLC_VISU
rounded rectangle at (60,230)-(91,251): text "%.1f"; shows WORD_TO_REAL(CronEd.PR.Setpoint[0])/10; runs INTERN ASSIGN CronEd.PR.Setpoint[0]:=(REAL_TO_WORD(CronEd.PR_TT*10))
rounded rectangle at (60,250)-(91,271): text "%.1f"; shows WORD_TO_REAL(CronEd.PR.Setpoint[1])/10; runs INTERN ASSIGN CronEd.PR.Setpoint[1]:=(REAL_TO_WORD(CronEd.PR_TT*10))
rounded rectangle at (60,270)-(91,291): text "%.1f"; shows WORD_TO_REAL(CronEd.PR.Setpoint[2])/10; runs INTERN ASSIGN CronEd.PR.Setpoint[2]:=(REAL_TO_WORD(CronEd.PR_TT*10))
rounded rectangle at (60,290)-(91,311): text "%.1f"; shows WORD_TO_REAL(CronEd.PR.Setpoint[3])/10; runs INTERN ASSIGN CronEd.PR.Setpoint[3]:=(REAL_TO_WORD(CronEd.PR_TT*10))
rectangle at (60,200)-(91,221): text "h00"; runs INTERN ASSIGN CronEd.PR.Setpoint[0]:=(REAL_TO_WORD(CronEd.PR_TT*10));INTERN ASSIGN CronEd.PR.Setpoint[1]:=(REAL_TO_WORD(CronEd.PR_TT*10));INTERN ASSIGN CronEd.PR.Setpoint[2]:=(REAL_TO_WORD(CronEd.PR_TT*10));INTERN ASSIGN CronEd.PR.Setpoint[3]:=(REAL_TO_WORD(CronEd.PR_TT*10))
rounded rectangle at (90,230)-(121,251): text "%.1f"; shows WORD_TO_REAL(CronEd.PR.Setpoint[4])/10; runs INTERN ASSIGN CronEd.PR.Setpoint[4]:=(REAL_TO_WORD(CronEd.PR_TT*10))
rounded rectangle at (90,250)-(121,271): text "%.1f"; shows WORD_TO_REAL(CronEd.PR.Setpoint[5])/10; runs INTERN ASSIGN CronEd.PR.Setpoint[5]:=(REAL_TO_WORD(CronEd.PR_TT*10))
rounded rectangle at (90,270)-(121,291): text "%.1f"; shows WORD_TO_REAL(CronEd.PR.Setpoint[6])/10; runs INTERN ASSIGN CronEd.PR.Setpoint[6]:=(REAL_TO_WORD(CronEd.PR_TT*10))
rounded rectangle at (90,290)-(121,311): text "%.1f"; shows WORD_TO_REAL(CronEd.PR.Setpoint[7])/10; runs INTERN ASSIGN CronEd.PR.Setpoint[7]:=(REAL_TO_WORD(CronEd.PR_TT*10))
rectangle at (90,200)-(121,221): text "h01"; runs INTERN ASSIGN CronEd.PR.Setpoint[4]:=(REAL_TO_WORD(CronEd.PR_TT*10));INTERN ASSIGN CronEd.PR.Setpoint[5]:=(REAL_TO_WORD(CronEd.PR_TT*10));INTERN ASSIGN CronEd.PR.Setpoint[6]:=(REAL_TO_WORD(CronEd.PR_TT*10));INTERN ASSIGN CronEd.PR.Setpoint[7]:=(REAL_TO_WORD(CronEd.PR_TT*10))
rounded rectangle at (120,230)-(151,251): text "%.1f"; shows WORD_TO_REAL(CronEd.PR.Setpoint[8])/10; runs INTERN ASSIGN CronEd.PR.Setpoint[8]:=(REAL_TO_WORD(CronEd.PR_TT*10))
rounded rectangle at (120,250)-(151,271): text "%.1f"; shows WORD_TO_REAL(CronEd.PR.Setpoint[9])/10; runs INTERN ASSIGN CronEd.PR.Setpoint[9]:=(REAL_TO_WORD(CronEd.PR_TT*10))
rounded rectangle at (120,270)-(151,291): text "%.1f"; shows WORD_TO_REAL(CronEd.PR.Setpoint[10])/10; runs INTERN ASSIGN CronEd.PR.Setpoint[10]:=(REAL_TO_WORD(CronEd.PR_TT*10))
rounded rectangle at (120,290)-(151,311): text "%.1f"; shows WORD_TO_REAL(CronEd.PR.Setpoint[11])/10; runs INTERN ASSIGN CronEd.PR.Setpoint[11]:=(REAL_TO_WORD(CronEd.PR_TT*10))
rectangle at (120,200)-(151,221): text "h02"; runs INTERN ASSIGN CronEd.PR.Setpoint[8]:=(REAL_TO_WORD(CronEd.PR_TT*10));INTERN ASSIGN CronEd.PR.Setpoint[9]:=(REAL_TO_WORD(CronEd.PR_TT*10));INTERN ASSIGN CronEd.PR.Setpoint[10]:=(REAL_TO_WORD(CronEd.PR_TT*10));INTERN ASSIGN CronEd.PR.Setpoint[11]:=(REAL_TO_WORD(CronEd.PR_TT*10))
rounded rectangle at (150,230)-(181,251): text "%.1f"; shows WORD_TO_REAL(CronEd.PR.Setpoint[12])/10; runs INTERN ASSIGN CronEd.PR.Setpoint[12]:=(REAL_TO_WORD(CronEd.PR_TT*10))
rounded rectangle at (150,250)-(181,271): text "%.1f"; shows WORD_TO_REAL(CronEd.PR.Setpoint[13])/10; runs INTERN ASSIGN CronEd.PR.Setpoint[13]:=(REAL_TO_WORD(CronEd.PR_TT*10))
rounded rectangle at (150,270)-(181,291): text "%.1f"; shows WORD_TO_REAL(CronEd.PR.Setpoint[14])/10; runs INTERN ASSIGN CronEd.PR.Setpoint[14]:=(REAL_TO_WORD(CronEd.PR_TT*10))
rounded rectangle at (150,290)-(181,311): text "%.1f"; shows WORD_TO_REAL(CronEd.PR.Setpoint[15])/10; runs INTERN ASSIGN CronEd.PR.Setpoint[15]:=(REAL_TO_WORD(CronEd.PR_TT*10))
rectangle at (150,200)-(181,221): text "h03"; runs INTERN ASSIGN CronEd.PR.Setpoint[15]:=(REAL_TO_WORD(CronEd.PR_TT*10));INTERN ASSIGN CronEd.PR.Setpoint[14]:=(REAL_TO_WORD(CronEd.PR_TT*10));INTERN ASSIGN CronEd.PR.Setpoint[13]:=(REAL_TO_WORD(CronEd.PR_TT*10));INTERN ASSIGN CronEd.PR.Setpoint[12]:=(REAL_TO_WORD(CronEd.PR_TT*10))
rounded rectangle at (180,230)-(211,251): text "%.1f"; shows WORD_TO_REAL(CronEd.PR.Setpoint[16])/10; runs INTERN ASSIGN CronEd.PR.Setpoint[16]:=(REAL_TO_WORD(CronEd.PR_TT*10))
rounded rectangle at (180,250)-(211,271): text "%.1f"; shows WORD_TO_REAL(CronEd.PR.Setpoint[17])/10; runs INTERN ASSIGN CronEd.PR.Setpoint[17]:=(REAL_TO_WORD(CronEd.PR_TT*10))
rounded rectangle at (180,270)-(211,291): text "%.1f"; shows WORD_TO_REAL(CronEd.PR.Setpoint[18])/10; runs INTERN ASSIGN CronEd.PR.Setpoint[18]:=(REAL_TO_WORD(CronEd.PR_TT*10))
rounded rectangle at (180,290)-(211,311): text "%.1f"; shows WORD_TO_REAL(CronEd.PR.Setpoint[19])/10; runs INTERN ASSIGN CronEd.PR.Setpoint[19]:=(REAL_TO_WORD(CronEd.PR_TT*10))
rectangle at (180,200)-(211,221): text "h04"; runs INTERN ASSIGN CronEd.PR.Setpoint[19]:=(REAL_TO_WORD(CronEd.PR_TT*10));INTERN ASSIGN CronEd.PR.Setpoint[18]:=(REAL_TO_WORD(CronEd.PR_TT*10));INTERN ASSIGN CronEd.PR.Setpoint[17]:=(REAL_TO_WORD(CronEd.PR_TT*10));INTERN ASSIGN CronEd.PR.Setpoint[16]:=(REAL_TO_WORD(CronEd.PR_TT*10))
rounded rectangle at (210,230)-(241,251): text "%.1f"; shows WORD_TO_REAL(CronEd.PR.Setpoint[20])/10; runs INTERN ASSIGN CronEd.PR.Setpoint[20]:=(REAL_TO_WORD(CronEd.PR_TT*10))
rounded rectangle at (210,250)-(241,271): text "%.1f"; shows WORD_TO_REAL(CronEd.PR.Setpoint[21])/10; runs INTERN ASSIGN CronEd.PR.Setpoint[21]:=(REAL_TO_WORD(CronEd.PR_TT*10))
rounded rectangle at (210,270)-(241,291): text "%.1f"; shows WORD_TO_REAL(CronEd.PR.Setpoint[22])/10; runs INTERN ASSIGN CronEd.PR.Setpoint[22]:=(REAL_TO_WORD(CronEd.PR_TT*10))
rounded rectangle at (210,290)-(241,311): text "%.1f"; shows WORD_TO_REAL(CronEd.PR.Setpoint[23])/10; runs INTERN ASSIGN CronEd.PR.Setpoint[23]:=(REAL_TO_WORD(CronEd.PR_TT*10))
rectangle at (210,200)-(241,221): text "h05"; runs INTERN ASSIGN CronEd.PR.Setpoint[23]:=(REAL_TO_WORD(CronEd.PR_TT*10));INTERN ASSIGN CronEd.PR.Setpoint[22]:=(REAL_TO_WORD(CronEd.PR_TT*10));INTERN ASSIGN CronEd.PR.Setpoint[21]:=(REAL_TO_WORD(CronEd.PR_TT*10));INTERN ASSIGN CronEd.PR.Setpoint[20]:=(REAL_TO_WORD(CronEd.PR_TT*10))
rounded rectangle at (240,230)-(271,251): text "%.1f"; shows WORD_TO_REAL(CronEd.PR.Setpoint[24])/10; runs INTERN ASSIGN CronEd.PR.Setpoint[24]:=(REAL_TO_WORD(CronEd.PR_TT*10))
rounded rectangle at (240,250)-(271,271): text "%.1f"; shows WORD_TO_REAL(CronEd.PR.Setpoint[25])/10; runs INTERN ASSIGN CronEd.PR.Setpoint[25]:=(REAL_TO_WORD(CronEd.PR_TT*10))
rounded rectangle at (240,270)-(271,291): text "%.1f"; shows WORD_TO_REAL(CronEd.PR.Setpoint[26])/10; runs INTERN ASSIGN CronEd.PR.Setpoint[26]:=(REAL_TO_WORD(CronEd.PR_TT*10))
rounded rectangle at (240,290)-(271,311): text "%.1f"; shows WORD_TO_REAL(CronEd.PR.Setpoint[27])/10; runs INTERN ASSIGN CronEd.PR.Setpoint[27]:=(REAL_TO_WORD(CronEd.PR_TT*10))
rectangle at (240,200)-(271,221): text "h06"; runs INTERN ASSIGN CronEd.PR.Setpoint[27]:=(REAL_TO_WORD(CronEd.PR_TT*10));INTERN ASSIGN CronEd.PR.Setpoint[26]:=(REAL_TO_WORD(CronEd.PR_TT*10));INTERN ASSIGN CronEd.PR.Setpoint[25]:=(REAL_TO_WORD(CronEd.PR_TT*10));INTERN ASSIGN CronEd.PR.Setpoint[24]:=(REAL_TO_WORD(CronEd.PR_TT*10))
rounded rectangle at (270,230)-(301,251): text "%.1f"; shows WORD_TO_REAL(CronEd.PR.Setpoint[28])/10; runs INTERN ASSIGN CronEd.PR.Setpoint[28]:=(REAL_TO_WORD(CronEd.PR_TT*10))
rounded rectangle at (270,250)-(301,271): text "%.1f"; shows WORD_TO_REAL(CronEd.PR.Setpoint[29])/10; runs INTERN ASSIGN CronEd.PR.Setpoint[29]:=(REAL_TO_WORD(CronEd.PR_TT*10))
rounded rectangle at (270,270)-(301,291): text "%.1f"; shows WORD_TO_REAL(CronEd.PR.Setpoint[30])/10; runs INTERN ASSIGN CronEd.PR.Setpoint[30]:=(REAL_TO_WORD(CronEd.PR_TT*10))
rounded rectangle at (270,290)-(301,311): text "%.1f"; shows WORD_TO_REAL(CronEd.PR.Setpoint[31])/10; runs INTERN ASSIGN CronEd.PR.Setpoint[31]:=(REAL_TO_WORD(CronEd.PR_TT*10))
rectangle at (270,200)-(301,221): text "h07"; runs INTERN ASSIGN CronEd.PR.Setpoint[31]:=(REAL_TO_WORD(CronEd.PR_TT*10));INTERN ASSIGN CronEd.PR.Setpoint[30]:=(REAL_TO_WORD(CronEd.PR_TT*10));INTERN ASSIGN CronEd.PR.Setpoint[29]:=(REAL_TO_WORD(CronEd.PR_TT*10));INTERN ASSIGN CronEd.PR.Setpoint[28]:=(REAL_TO_WORD(CronEd.PR_TT*10))
rounded rectangle at (300,230)-(331,251): text "%.1f"; shows WORD_TO_REAL(CronEd.PR.Setpoint[32])/10; runs INTERN ASSIGN CronEd.PR.Setpoint[32]:=(REAL_TO_WORD(CronEd.PR_TT*10))
rounded rectangle at (300,250)-(331,271): text "%.1f"; shows WORD_TO_REAL(CronEd.PR.Setpoint[33])/10; runs INTERN ASSIGN CronEd.PR.Setpoint[33]:=(REAL_TO_WORD(CronEd.PR_TT*10))
rounded rectangle at (300,270)-(331,291): text "%.1f"; shows WORD_TO_REAL(CronEd.PR.Setpoint[34])/10; runs INTERN ASSIGN CronEd.PR.Setpoint[34]:=(REAL_TO_WORD(CronEd.PR_TT*10))
rounded rectangle at (300,290)-(331,311): text "%.1f"; shows WORD_TO_REAL(CronEd.PR.Setpoint[35])/10; runs INTERN ASSIGN CronEd.PR.Setpoint[35]:=(REAL_TO_WORD(CronEd.PR_TT*10))
rectangle at (300,200)-(331,221): text "h08"; runs INTERN ASSIGN CronEd.PR.Setpoint[35]:=(REAL_TO_WORD(CronEd.PR_TT*10));INTERN ASSIGN CronEd.PR.Setpoint[34]:=(REAL_TO_WORD(CronEd.PR_TT*10));INTERN ASSIGN CronEd.PR.Setpoint[33]:=(REAL_TO_WORD(CronEd.PR_TT*10));INTERN ASSIGN CronEd.PR.Setpoint[32]:=(REAL_TO_WORD(CronEd.PR_TT*10))
rounded rectangle at (330,230)-(361,251): text "%.1f"; shows WORD_TO_REAL(CronEd.PR.Setpoint[36])/10; runs INTERN ASSIGN CronEd.PR.Setpoint[36]:=(REAL_TO_WORD(CronEd.PR_TT*10))
rounded rectangle at (330,250)-(361,271): text "%.1f"; shows WORD_TO_REAL(CronEd.PR.Setpoint[37])/10; runs INTERN ASSIGN CronEd.PR.Setpoint[37]:=(REAL_TO_WORD(CronEd.PR_TT*10))
rounded rectangle at (330,270)-(361,291): text "%.1f"; shows WORD_TO_REAL(CronEd.PR.Setpoint[38])/10; runs INTERN ASSIGN CronEd.PR.Setpoint[38]:=(REAL_TO_WORD(CronEd.PR_TT*10))
rounded rectangle at (330,290)-(361,311): text "%.1f"; shows WORD_TO_REAL(CronEd.PR.Setpoint[39])/10; runs INTERN ASSIGN CronEd.PR.Setpoint[39]:=(REAL_TO_WORD(CronEd.PR_TT*10))
rectangle at (330,200)-(361,221): text "h09"; runs INTERN ASSIGN CronEd.PR.Setpoint[39]:=(REAL_TO_WORD(CronEd.PR_TT*10));INTERN ASSIGN CronEd.PR.Setpoint[38]:=(REAL_TO_WORD(CronEd.PR_TT*10));INTERN ASSIGN CronEd.PR.Setpoint[37]:=(REAL_TO_WORD(CronEd.PR_TT*10));INTERN ASSIGN CronEd.PR.Setpoint[36]:=(REAL_TO_WORD(CronEd.PR_TT*10))
rounded rectangle at (360,230)-(391,251): text "%.1f"; shows WORD_TO_REAL(CronEd.PR.Setpoint[40])/10; runs INTERN ASSIGN CronEd.PR.Setpoint[40]:=(REAL_TO_WORD(CronEd.PR_TT*10))
rounded rectangle at (360,250)-(391,271): text "%.1f"; shows WORD_TO_REAL(CronEd.PR.Setpoint[41])/10; runs INTERN ASSIGN CronEd.PR.Setpoint[41]:=(REAL_TO_WORD(CronEd.PR_TT*10))
rounded rectangle at (360,270)-(391,291): text "%.1f"; shows WORD_TO_REAL(CronEd.PR.Setpoint[42])/10; runs INTERN ASSIGN CronEd.PR.Setpoint[42]:=(REAL_TO_WORD(CronEd.PR_TT*10))
rounded rectangle at (360,290)-(391,311): text "%.1f"; shows WORD_TO_REAL(CronEd.PR.Setpoint[43])/10; runs INTERN ASSIGN CronEd.PR.Setpoint[43]:=(REAL_TO_WORD(CronEd.PR_TT*10))
rectangle at (360,200)-(391,221): text "h10"; runs INTERN ASSIGN CronEd.PR.Setpoint[43]:=(REAL_TO_WORD(CronEd.PR_TT*10));INTERN ASSIGN CronEd.PR.Setpoint[42]:=(REAL_TO_WORD(CronEd.PR_TT*10));INTERN ASSIGN CronEd.PR.Setpoint[41]:=(REAL_TO_WORD(CronEd.PR_TT*10));INTERN ASSIGN CronEd.PR.Setpoint[40]:=(REAL_TO_WORD(CronEd.PR_TT*10))
rounded rectangle at (390,230)-(421,251): text "%.1f"; shows WORD_TO_REAL(CronEd.PR.Setpoint[44])/10; runs INTERN ASSIGN CronEd.PR.Setpoint[44]:=(REAL_TO_WORD(CronEd.PR_TT*10))
rounded rectangle at (390,250)-(421,271): text "%.1f"; shows WORD_TO_REAL(CronEd.PR.Setpoint[45])/10; runs INTERN ASSIGN CronEd.PR.Setpoint[45]:=(REAL_TO_WORD(CronEd.PR_TT*10))
rounded rectangle at (390,270)-(421,291): text "%.1f"; shows WORD_TO_REAL(CronEd.PR.Setpoint[46])/10; runs INTERN ASSIGN CronEd.PR.Setpoint[46]:=(REAL_TO_WORD(CronEd.PR_TT*10))
rounded rectangle at (390,290)-(421,311): text "%.1f"; shows WORD_TO_REAL(CronEd.PR.Setpoint[47])/10; runs INTERN ASSIGN CronEd.PR.Setpoint[47]:=(REAL_TO_WORD(CronEd.PR_TT*10))
rectangle at (390,200)-(421,221): text "h11"; runs INTERN ASSIGN CronEd.PR.Setpoint[47]:=(REAL_TO_WORD(CronEd.PR_TT*10));INTERN ASSIGN CronEd.PR.Setpoint[46]:=(REAL_TO_WORD(CronEd.PR_TT*10));INTERN ASSIGN CronEd.PR.Setpoint[45]:=(REAL_TO_WORD(CronEd.PR_TT*10));INTERN ASSIGN CronEd.PR.Setpoint[44]:=(REAL_TO_WORD(CronEd.PR_TT*10))
rounded rectangle at (420,230)-(451,251): text "%.1f"; shows WORD_TO_REAL(CronEd.PR.Setpoint[48])/10; runs INTERN ASSIGN CronEd.PR.Setpoint[48]:=(REAL_TO_WORD(CronEd.PR_TT*10))
rounded rectangle at (420,250)-(451,271): text "%.1f"; shows WORD_TO_REAL(CronEd.PR.Setpoint[49])/10; runs INTERN ASSIGN CronEd.PR.Setpoint[49]:=(REAL_TO_WORD(CronEd.PR_TT*10))
rounded rectangle at (420,270)-(451,291): text "%.1f"; shows WORD_TO_REAL(CronEd.PR.Setpoint[50])/10; runs INTERN ASSIGN CronEd.PR.Setpoint[50]:=(REAL_TO_WORD(CronEd.PR_TT*10))
rounded rectangle at (420,290)-(451,311): text "%.1f"; shows WORD_TO_REAL(CronEd.PR.Setpoint[51])/10; runs INTERN ASSIGN CronEd.PR.Setpoint[51]:=(REAL_TO_WORD(CronEd.PR_TT*10))
rectangle at (420,200)-(451,221): text "h12"; runs INTERN ASSIGN CronEd.PR.Setpoint[51]:=(REAL_TO_WORD(CronEd.PR_TT*10));INTERN ASSIGN CronEd.PR.Setpoint[50]:=(REAL_TO_WORD(CronEd.PR_TT*10));INTERN ASSIGN CronEd.PR.Setpoint[49]:=(REAL_TO_WORD(CronEd.PR_TT*10));INTERN ASSIGN CronEd.PR.Setpoint[48]:=(REAL_TO_WORD(CronEd.PR_TT*10))
rounded rectangle at (450,230)-(481,251): text "%.1f"; shows WORD_TO_REAL(CronEd.PR.Setpoint[52])/10; runs INTERN ASSIGN CronEd.PR.Setpoint[52]:=(REAL_TO_WORD(CronEd.PR_TT*10))
rounded rectangle at (450,250)-(481,271): text "%.1f"; shows WORD_TO_REAL(CronEd.PR.Setpoint[53])/10; runs INTERN ASSIGN CronEd.PR.Setpoint[53]:=(REAL_TO_WORD(CronEd.PR_TT*10))
rounded rectangle at (450,270)-(481,291): text "%.1f"; shows WORD_TO_REAL(CronEd.PR.Setpoint[54])/10; runs INTERN ASSIGN CronEd.PR.Setpoint[54]:=(REAL_TO_WORD(CronEd.PR_TT*10))
rounded rectangle at (450,290)-(481,311): text "%.1f"; shows WORD_TO_REAL(CronEd.PR.Setpoint[55])/10; runs INTERN ASSIGN CronEd.PR.Setpoint[55]:=(REAL_TO_WORD(CronEd.PR_TT*10))
rectangle at (450,200)-(481,221): text "h13"; runs INTERN ASSIGN CronEd.PR.Setpoint[55]:=(REAL_TO_WORD(CronEd.PR_TT*10));INTERN ASSIGN CronEd.PR.Setpoint[54]:=(REAL_TO_WORD(CronEd.PR_TT*10));INTERN ASSIGN CronEd.PR.Setpoint[53]:=(REAL_TO_WORD(CronEd.PR_TT*10));INTERN ASSIGN CronEd.PR.Setpoint[52]:=(REAL_TO_WORD(CronEd.PR_TT*10))
rounded rectangle at (480,230)-(511,251): text "%.1f"; shows WORD_TO_REAL(CronEd.PR.Setpoint[56])/10; runs INTERN ASSIGN CronEd.PR.Setpoint[56]:=(REAL_TO_WORD(CronEd.PR_TT*10))
rounded rectangle at (480,250)-(511,271): text "%.1f"; shows WORD_TO_REAL(CronEd.PR.Setpoint[57])/10; runs INTERN ASSIGN CronEd.PR.Setpoint[57]:=(REAL_TO_WORD(CronEd.PR_TT*10))
rounded rectangle at (480,270)-(511,291): text "%.1f"; shows WORD_TO_REAL(CronEd.PR.Setpoint[58])/10; runs INTERN ASSIGN CronEd.PR.Setpoint[58]:=(REAL_TO_WORD(CronEd.PR_TT*10))
rounded rectangle at (480,290)-(511,311): text "%.1f"; shows WORD_TO_REAL(CronEd.PR.Setpoint[59])/10; runs INTERN ASSIGN CronEd.PR.Setpoint[59]:=(REAL_TO_WORD(CronEd.PR_TT*10))
rectangle at (480,200)-(511,221): text "h14"; runs INTERN ASSIGN CronEd.PR.Setpoint[59]:=(REAL_TO_WORD(CronEd.PR_TT*10));INTERN ASSIGN CronEd.PR.Setpoint[58]:=(REAL_TO_WORD(CronEd.PR_TT*10));INTERN ASSIGN CronEd.PR.Setpoint[57]:=(REAL_TO_WORD(CronEd.PR_TT*10));INTERN ASSIGN CronEd.PR.Setpoint[56]:=(REAL_TO_WORD(CronEd.PR_TT*10))
rounded rectangle at (510,230)-(541,251): text "%.1f"; shows WORD_TO_REAL(CronEd.PR.Setpoint[60])/10; runs INTERN ASSIGN CronEd.PR.Setpoint[60]:=(REAL_TO_WORD(CronEd.PR_TT*10))
rounded rectangle at (510,250)-(541,271): text "%.1f"; shows WORD_TO_REAL(CronEd.PR.Setpoint[61])/10; runs INTERN ASSIGN CronEd.PR.Setpoint[61]:=(REAL_TO_WORD(CronEd.PR_TT*10))
rounded rectangle at (510,270)-(541,291): text "%.1f"; shows WORD_TO_REAL(CronEd.PR.Setpoint[62])/10; runs INTERN ASSIGN CronEd.PR.Setpoint[62]:=(REAL_TO_WORD(CronEd.PR_TT*10))
rounded rectangle at (510,290)-(541,311): text "%.1f"; shows WORD_TO_REAL(CronEd.PR.Setpoint[63])/10; runs INTERN ASSIGN CronEd.PR.Setpoint[63]:=(REAL_TO_WORD(CronEd.PR_TT*10))
rectangle at (510,200)-(541,221): text "h15"; runs INTERN ASSIGN CronEd.PR.Setpoint[63]:=(REAL_TO_WORD(CronEd.PR_TT*10));INTERN ASSIGN CronEd.PR.Setpoint[62]:=(REAL_TO_WORD(CronEd.PR_TT*10));INTERN ASSIGN CronEd.PR.Setpoint[61]:=(REAL_TO_WORD(CronEd.PR_TT*10));INTERN ASSIGN CronEd.PR.Setpoint[60]:=(REAL_TO_WORD(CronEd.PR_TT*10))
rounded rectangle at (540,230)-(571,251): text "%.1f"; shows WORD_TO_REAL(CronEd.PR.Setpoint[64])/10; runs INTERN ASSIGN CronEd.PR.Setpoint[64]:=(REAL_TO_WORD(CronEd.PR_TT*10))
rounded rectangle at (540,250)-(571,271): text "%.1f"; shows WORD_TO_REAL(CronEd.PR.Setpoint[65])/10; runs INTERN ASSIGN CronEd.PR.Setpoint[65]:=(REAL_TO_WORD(CronEd.PR_TT*10))
rounded rectangle at (540,270)-(571,291): text "%.1f"; shows WORD_TO_REAL(CronEd.PR.Setpoint[66])/10; runs INTERN ASSIGN CronEd.PR.Setpoint[66]:=(REAL_TO_WORD(CronEd.PR_TT*10))
rounded rectangle at (540,290)-(571,311): text "%.1f"; shows WORD_TO_REAL(CronEd.PR.Setpoint[67])/10; runs INTERN ASSIGN CronEd.PR.Setpoint[67]:=(REAL_TO_WORD(CronEd.PR_TT*10))
rectangle at (540,200)-(571,221): text "h16"; runs INTERN ASSIGN CronEd.PR.Setpoint[67]:=(REAL_TO_WORD(CronEd.PR_TT*10));INTERN ASSIGN CronEd.PR.Setpoint[66]:=(REAL_TO_WORD(CronEd.PR_TT*10));INTERN ASSIGN CronEd.PR.Setpoint[65]:=(REAL_TO_WORD(CronEd.PR_TT*10));INTERN ASSIGN CronEd.PR.Setpoint[64]:=(REAL_TO_WORD(CronEd.PR_TT*10))
rounded rectangle at (570,230)-(601,251): text "%.1f"; shows WORD_TO_REAL(CronEd.PR.Setpoint[68])/10; runs INTERN ASSIGN CronEd.PR.Setpoint[68]:=(REAL_TO_WORD(CronEd.PR_TT*10))
rounded rectangle at (570,250)-(601,271): text "%.1f"; shows WORD_TO_REAL(CronEd.PR.Setpoint[69])/10; runs INTERN ASSIGN CronEd.PR.Setpoint[69]:=(REAL_TO_WORD(CronEd.PR_TT*10))
rounded rectangle at (570,270)-(601,291): text "%.1f"; shows WORD_TO_REAL(CronEd.PR.Setpoint[70])/10; runs INTERN ASSIGN CronEd.PR.Setpoint[70]:=(REAL_TO_WORD(CronEd.PR_TT*10))
rounded rectangle at (570,290)-(601,311): text "%.1f"; shows WORD_TO_REAL(CronEd.PR.Setpoint[71])/10; runs INTERN ASSIGN CronEd.PR.Setpoint[71]:=(REAL_TO_WORD(CronEd.PR_TT*10))
rectangle at (570,200)-(601,221): text "h17"; runs INTERN ASSIGN CronEd.PR.Setpoint[71]:=(REAL_TO_WORD(CronEd.PR_TT*10));INTERN ASSIGN CronEd.PR.Setpoint[70]:=(REAL_TO_WORD(CronEd.PR_TT*10));INTERN ASSIGN CronEd.PR.Setpoint[69]:=(REAL_TO_WORD(CronEd.PR_TT*10));INTERN ASSIGN CronEd.PR.Setpoint[68]:=(REAL_TO_WORD(CronEd.PR_TT*10))
rounded rectangle at (600,230)-(631,251): text "%.1f"; shows WORD_TO_REAL(CronEd.PR.Setpoint[72])/10; runs INTERN ASSIGN CronEd.PR.Setpoint[72]:=(REAL_TO_WORD(CronEd.PR_TT*10))
rounded rectangle at (600,250)-(631,271): text "%.1f"; shows WORD_TO_REAL(CronEd.PR.Setpoint[73])/10; runs INTERN ASSIGN CronEd.PR.Setpoint[73]:=(REAL_TO_WORD(CronEd.PR_TT*10))
rounded rectangle at (600,270)-(631,291): text "%.1f"; shows WORD_TO_REAL(CronEd.PR.Setpoint[74])/10; runs INTERN ASSIGN CronEd.PR.Setpoint[74]:=(REAL_TO_WORD(CronEd.PR_TT*10))
rounded rectangle at (600,290)-(631,311): text "%.1f"; shows WORD_TO_REAL(CronEd.PR.Setpoint[75])/10; runs INTERN ASSIGN CronEd.PR.Setpoint[75]:=(REAL_TO_WORD(CronEd.PR_TT*10))
rectangle at (600,200)-(631,221): text "h18"; runs INTERN ASSIGN CronEd.PR.Setpoint[75]:=(REAL_TO_WORD(CronEd.PR_TT*10));INTERN ASSIGN CronEd.PR.Setpoint[74]:=(REAL_TO_WORD(CronEd.PR_TT*10));INTERN ASSIGN CronEd.PR.Setpoint[73]:=(REAL_TO_WORD(CronEd.PR_TT*10));INTERN ASSIGN CronEd.PR.Setpoint[72]:=(REAL_TO_WORD(CronEd.PR_TT*10))
rounded rectangle at (630,230)-(661,251): text "%.1f"; shows WORD_TO_REAL(CronEd.PR.Setpoint[76])/10; runs INTERN ASSIGN CronEd.PR.Setpoint[76]:=(REAL_TO_WORD(CronEd.PR_TT*10))
rounded rectangle at (630,250)-(661,271): text "%.1f"; shows WORD_TO_REAL(CronEd.PR.Setpoint[77])/10; runs INTERN ASSIGN CronEd.PR.Setpoint[77]:=(REAL_TO_WORD(CronEd.PR_TT*10))
rounded rectangle at (630,270)-(661,291): text "%.1f"; shows WORD_TO_REAL(CronEd.PR.Setpoint[78])/10; runs INTERN ASSIGN CronEd.PR.Setpoint[78]:=(REAL_TO_WORD(CronEd.PR_TT*10))
rounded rectangle at (630,290)-(661,311): text "%.1f"; shows WORD_TO_REAL(CronEd.PR.Setpoint[79])/10; runs INTERN ASSIGN CronEd.PR.Setpoint[79]:=(REAL_TO_WORD(CronEd.PR_TT*10))
rectangle at (630,200)-(661,221): text "h19"; runs INTERN ASSIGN CronEd.PR.Setpoint[79]:=(REAL_TO_WORD(CronEd.PR_TT*10));INTERN ASSIGN CronEd.PR.Setpoint[78]:=(REAL_TO_WORD(CronEd.PR_TT*10));INTERN ASSIGN CronEd.PR.Setpoint[77]:=(REAL_TO_WORD(CronEd.PR_TT*10));INTERN ASSIGN CronEd.PR.Setpoint[76]:=(REAL_TO_WORD(CronEd.PR_TT*10))
rounded rectangle at (660,230)-(691,251): text "%.1f"; shows WORD_TO_REAL(CronEd.PR.Setpoint[80])/10; runs INTERN ASSIGN CronEd.PR.Setpoint[80]:=(REAL_TO_WORD(CronEd.PR_TT*10))
rounded rectangle at (660,250)-(691,271): text "%.1f"; shows WORD_TO_REAL(CronEd.PR.Setpoint[81])/10; runs INTERN ASSIGN CronEd.PR.Setpoint[81]:=(REAL_TO_WORD(CronEd.PR_TT*10))
rounded rectangle at (660,270)-(691,291): text "%.1f"; shows WORD_TO_REAL(CronEd.PR.Setpoint[82])/10; runs INTERN ASSIGN CronEd.PR.Setpoint[82]:=(REAL_TO_WORD(CronEd.PR_TT*10))
rounded rectangle at (660,290)-(691,311): text "%.1f"; shows WORD_TO_REAL(CronEd.PR.Setpoint[83])/10; runs INTERN ASSIGN CronEd.PR.Setpoint[83]:=(REAL_TO_WORD(CronEd.PR_TT*10))
rectangle at (660,200)-(691,221): text "h20"; runs INTERN ASSIGN CronEd.PR.Setpoint[83]:=(REAL_TO_WORD(CronEd.PR_TT*10));INTERN ASSIGN CronEd.PR.Setpoint[82]:=(REAL_TO_WORD(CronEd.PR_TT*10));INTERN ASSIGN CronEd.PR.Setpoint[81]:=(REAL_TO_WORD(CronEd.PR_TT*10));INTERN ASSIGN CronEd.PR.Setpoint[80]:=(REAL_TO_WORD(CronEd.PR_TT*10))
rounded rectangle at (690,230)-(721,251): text "%.1f"; shows WORD_TO_REAL(CronEd.PR.Setpoint[84])/10; runs INTERN ASSIGN CronEd.PR.Setpoint[84]:=(REAL_TO_WORD(CronEd.PR_TT*10))
rounded rectangle at (690,250)-(721,271): text "%.1f"; shows WORD_TO_REAL(CronEd.PR.Setpoint[85])/10; runs INTERN ASSIGN CronEd.PR.Setpoint[85]:=(REAL_TO_WORD(CronEd.PR_TT*10))
rounded rectangle at (690,270)-(721,291): text "%.1f"; shows WORD_TO_REAL(CronEd.PR.Setpoint[86])/10; runs INTERN ASSIGN CronEd.PR.Setpoint[86]:=(REAL_TO_WORD(CronEd.PR_TT*10))
rounded rectangle at (690,290)-(721,311): text "%.1f"; shows WORD_TO_REAL(CronEd.PR.Setpoint[87])/10; runs INTERN ASSIGN CronEd.PR.Setpoint[87]:=(REAL_TO_WORD(CronEd.PR_TT*10))
rectangle at (690,200)-(721,221): text "h21"; runs INTERN ASSIGN CronEd.PR.Setpoint[87]:=(REAL_TO_WORD(CronEd.PR_TT*10));INTERN ASSIGN CronEd.PR.Setpoint[86]:=(REAL_TO_WORD(CronEd.PR_TT*10));INTERN ASSIGN CronEd.PR.Setpoint[85]:=(REAL_TO_WORD(CronEd.PR_TT*10));INTERN ASSIGN CronEd.PR.Setpoint[84]:=(REAL_TO_WORD(CronEd.PR_TT*10))
rounded rectangle at (720,230)-(751,251): text "%.1f"; shows WORD_TO_REAL(CronEd.PR.Setpoint[88])/10; runs INTERN ASSIGN CronEd.PR.Setpoint[88]:=(REAL_TO_WORD(CronEd.PR_TT*10))
rounded rectangle at (720,250)-(751,271): text "%.1f"; shows WORD_TO_REAL(CronEd.PR.Setpoint[89])/10; runs INTERN ASSIGN CronEd.PR.Setpoint[89]:=(REAL_TO_WORD(CronEd.PR_TT*10))
rounded rectangle at (720,270)-(751,291): text "%.1f"; shows WORD_TO_REAL(CronEd.PR.Setpoint[90])/10; runs INTERN ASSIGN CronEd.PR.Setpoint[90]:=(REAL_TO_WORD(CronEd.PR_TT*10))
rounded rectangle at (720,290)-(751,311): text "%.1f"; shows WORD_TO_REAL(CronEd.PR.Setpoint[91])/10; runs INTERN ASSIGN CronEd.PR.Setpoint[91]:=(REAL_TO_WORD(CronEd.PR_TT*10))
rectangle at (720,200)-(751,221): text "h22"; runs INTERN ASSIGN CronEd.PR.Setpoint[91]:=(REAL_TO_WORD(CronEd.PR_TT*10));INTERN ASSIGN CronEd.PR.Setpoint[90]:=(REAL_TO_WORD(CronEd.PR_TT*10));INTERN ASSIGN CronEd.PR.Setpoint[89]:=(REAL_TO_WORD(CronEd.PR_TT*10));INTERN ASSIGN CronEd.PR.Setpoint[88]:=(REAL_TO_WORD(CronEd.PR_TT*10))
rounded rectangle at (750,230)-(781,251): text "%.1f"; shows WORD_TO_REAL(CronEd.PR.Setpoint[92])/10; runs INTERN ASSIGN CronEd.PR.Setpoint[92]:=(REAL_TO_WORD(CronEd.PR_TT*10))
rounded rectangle at (750,250)-(781,271): text "%.1f"; shows WORD_TO_REAL(CronEd.PR.Setpoint[93])/10; runs INTERN ASSIGN CronEd.PR.Setpoint[93]:=(REAL_TO_WORD(CronEd.PR_TT*10))
rounded rectangle at (750,270)-(781,291): text "%.1f"; shows WORD_TO_REAL(CronEd.PR.Setpoint[94])/10; runs INTERN ASSIGN CronEd.PR.Setpoint[94]:=(REAL_TO_WORD(CronEd.PR_TT*10))
rounded rectangle at (750,290)-(781,311): text "%.1f"; shows WORD_TO_REAL(CronEd.PR.Setpoint[95])/10; runs INTERN ASSIGN CronEd.PR.Setpoint[95]:=(REAL_TO_WORD(CronEd.PR_TT*10))
rectangle at (750,200)-(781,221): text "h23"; runs INTERN ASSIGN CronEd.PR.Setpoint[95]:=(REAL_TO_WORD(CronEd.PR_TT*10));INTERN ASSIGN CronEd.PR.Setpoint[94]:=(REAL_TO_WORD(CronEd.PR_TT*10));INTERN ASSIGN CronEd.PR.Setpoint[93]:=(REAL_TO_WORD(CronEd.PR_TT*10));INTERN ASSIGN CronEd.PR.Setpoint[92]:=(REAL_TO_WORD(CronEd.PR_TT*10))
rectangle at (410,360)-(491,381): text "Month"
rectangle at (490,360)-(531,381): text "%d"; shows CronEd.CA_Sel; alarm colour if CronEd.CA_Sel<>CronEd.CA_Act; editable 1..12
rectangle at (410,390)-(491,411): text "Profile Nr."
rectangle at (490,390)-(531,411): text "%d"; shows CronEd.CA_TPR; editable 0..10
button at (540,360)-(601,381): text "Load"; toggles CronEd.CA_Load
button at (610,360)-(671,381): text "Save"; toggles CronEd.CA_Save
rounded rectangle at (160,360)-(191,381): text "%d"; shows CronEd.CA.Profile[0]; invisible if CronEd.CA_DayF>0; alarm colour if CronEd.CA.Profile[0]=0; runs INTERN ASSIGN CronEd.CA.Profile[0]:=(CronEd.CA_TPR)
rectangle at (120,360)-(151,381): text "1"
rounded rectangle at (190,360)-(221,381): text "%d"; shows CronEd.CA.Profile[1]; invisible if CronEd.CA_DayF>1; alarm colour if CronEd.CA.Profile[1]=0; runs INTERN ASSIGN CronEd.CA.Profile[1]:=(CronEd.CA_TPR)
rounded rectangle at (220,360)-(251,381): text "%d"; shows CronEd.CA.Profile[2]; invisible if CronEd.CA_DayF>2; alarm colour if CronEd.CA.Profile[2]=0; runs INTERN ASSIGN CronEd.CA.Profile[2]:=(CronEd.CA_TPR)
rounded rectangle at (250,360)-(281,381): text "%d"; shows CronEd.CA.Profile[3]; invisible if CronEd.CA_DayF>3; alarm colour if CronEd.CA.Profile[3]=0; runs INTERN ASSIGN CronEd.CA.Profile[3]:=(CronEd.CA_TPR)
rounded rectangle at (280,360)-(311,381): text "%d"; shows CronEd.CA.Profile[4]; invisible if CronEd.CA_DayF>4; alarm colour if CronEd.CA.Profile[4]=0; runs INTERN ASSIGN CronEd.CA.Profile[4]:=(CronEd.CA_TPR)
rounded rectangle at (310,360)-(341,381): text "%d"; shows CronEd.CA.Profile[5]; invisible if CronEd.CA_DayF>5; alarm colour if CronEd.CA.Profile[5]=0; runs INTERN ASSIGN CronEd.CA.Profile[5]:=(CronEd.CA_TPR)
rounded rectangle at (340,360)-(371,381): text "%d"; shows CronEd.CA.Profile[6]; alarm colour if CronEd.CA.Profile[6]=0; runs INTERN ASSIGN CronEd.CA.Profile[6]:=(CronEd.CA_TPR)
rounded rectangle at (160,380)-(191,401): text "%d"; shows CronEd.CA.Profile[7]; alarm colour if CronEd.CA.Profile[7]=0; runs INTERN ASSIGN CronEd.CA.Profile[7]:=(CronEd.CA_TPR)
rectangle at (120,380)-(151,401): text "8"
rounded rectangle at (190,380)-(221,401): text "%d"; shows CronEd.CA.Profile[8]; alarm colour if CronEd.CA.Profile[8]=0; runs INTERN ASSIGN CronEd.CA.Profile[8]:=(CronEd.CA_TPR)
rounded rectangle at (220,380)-(251,401): text "%d"; shows CronEd.CA.Profile[9]; alarm colour if CronEd.CA.Profile[9]=0; runs INTERN ASSIGN CronEd.CA.Profile[9]:=(CronEd.CA_TPR)
rounded rectangle at (250,380)-(281,401): text "%d"; shows CronEd.CA.Profile[10]; alarm colour if CronEd.CA.Profile[10]=0; runs INTERN ASSIGN CronEd.CA.Profile[10]:=(CronEd.CA_TPR)
rounded rectangle at (280,380)-(311,401): text "%d"; shows CronEd.CA.Profile[11]; alarm colour if CronEd.CA.Profile[11]=0; runs INTERN ASSIGN CronEd.CA.Profile[11]:=(CronEd.CA_TPR)
rounded rectangle at (310,380)-(341,401): text "%d"; shows CronEd.CA.Profile[12]; alarm colour if CronEd.CA.Profile[12]=0; runs INTERN ASSIGN CronEd.CA.Profile[12]:=(CronEd.CA_TPR)
rounded rectangle at (340,380)-(371,401): text "%d"; shows CronEd.CA.Profile[13]; alarm colour if CronEd.CA.Profile[13]=0; runs INTERN ASSIGN CronEd.CA.Profile[13]:=(CronEd.CA_TPR)
rounded rectangle at (160,400)-(191,421): text "%d"; shows CronEd.CA.Profile[14]; alarm colour if CronEd.CA.Profile[14]=0; runs INTERN ASSIGN CronEd.CA.Profile[14]:=(CronEd.CA_TPR)
rectangle at (120,400)-(151,421): text "15"
rounded rectangle at (190,400)-(221,421): text "%d"; shows CronEd.CA.Profile[15]; alarm colour if CronEd.CA.Profile[15]=0; runs INTERN ASSIGN CronEd.CA.Profile[15]:=(CronEd.CA_TPR)
rounded rectangle at (220,400)-(251,421): text "%d"; shows CronEd.CA.Profile[16]; alarm colour if CronEd.CA.Profile[16]=0; runs INTERN ASSIGN CronEd.CA.Profile[16]:=(CronEd.CA_TPR)
rounded rectangle at (250,400)-(281,421): text "%d"; shows CronEd.CA.Profile[17]; alarm colour if CronEd.CA.Profile[17]=0; runs INTERN ASSIGN CronEd.CA.Profile[17]:=(CronEd.CA_TPR)
rounded rectangle at (280,400)-(311,421): text "%d"; shows CronEd.CA.Profile[18]; alarm colour if CronEd.CA.Profile[18]=0; runs INTERN ASSIGN CronEd.CA.Profile[18]:=(CronEd.CA_TPR)
rounded rectangle at (310,400)-(341,421): text "%d"; shows CronEd.CA.Profile[19]; alarm colour if CronEd.CA.Profile[19]=0; runs INTERN ASSIGN CronEd.CA.Profile[19]:=(CronEd.CA_TPR)
rounded rectangle at (340,400)-(371,421): text "%d"; shows CronEd.CA.Profile[20]; alarm colour if CronEd.CA.Profile[20]=0; runs INTERN ASSIGN CronEd.CA.Profile[20]:=(CronEd.CA_TPR)
rounded rectangle at (160,420)-(191,441): text "%d"; shows CronEd.CA.Profile[21]; alarm colour if CronEd.CA.Profile[21]=0; runs INTERN ASSIGN CronEd.CA.Profile[21]:=(CronEd.CA_TPR)
rectangle at (120,420)-(151,441): text "22"
rounded rectangle at (190,420)-(221,441): text "%d"; shows CronEd.CA.Profile[22]; alarm colour if CronEd.CA.Profile[22]=0; runs INTERN ASSIGN CronEd.CA.Profile[22]:=(CronEd.CA_TPR)
rounded rectangle at (220,420)-(251,441): text "%d"; shows CronEd.CA.Profile[23]; alarm colour if CronEd.CA.Profile[23]=0; runs INTERN ASSIGN CronEd.CA.Profile[23]:=(CronEd.CA_TPR)
rounded rectangle at (250,420)-(281,441): text "%d"; shows CronEd.CA.Profile[24]; alarm colour if CronEd.CA.Profile[24]=0; runs INTERN ASSIGN CronEd.CA.Profile[24]:=(CronEd.CA_TPR)
rounded rectangle at (280,420)-(311,441): text "%d"; shows CronEd.CA.Profile[25]; alarm colour if CronEd.CA.Profile[25]=0; runs INTERN ASSIGN CronEd.CA.Profile[25]:=(CronEd.CA_TPR)
rounded rectangle at (310,420)-(341,441): text "%d"; shows CronEd.CA.Profile[26]; alarm colour if CronEd.CA.Profile[26]=0; runs INTERN ASSIGN CronEd.CA.Profile[26]:=(CronEd.CA_TPR)
rounded rectangle at (340,420)-(371,441): text "%d"; shows CronEd.CA.Profile[27]; alarm colour if CronEd.CA.Profile[27]=0; runs INTERN ASSIGN CronEd.CA.Profile[27]:=(CronEd.CA_TPR)
rounded rectangle at (160,440)-(191,461): text "%d"; shows CronEd.CA.Profile[28]; alarm colour if CronEd.CA.Profile[28]=0; runs INTERN ASSIGN CronEd.CA.Profile[28]:=(CronEd.CA_TPR)
rectangle at (120,440)-(151,461): text "29"
rounded rectangle at (190,440)-(221,461): text "%d"; shows CronEd.CA.Profile[29]; alarm colour if CronEd.CA.Profile[29]=0; runs INTERN ASSIGN CronEd.CA.Profile[29]:=(CronEd.CA_TPR)
rounded rectangle at (220,440)-(251,461): text "%d"; shows CronEd.CA.Profile[30]; alarm colour if CronEd.CA.Profile[30]=0; runs INTERN ASSIGN CronEd.CA.Profile[30]:=(CronEd.CA_TPR)
rounded rectangle at (250,440)-(281,461): text "%d"; shows CronEd.CA.Profile[31]; alarm colour if CronEd.CA.Profile[31]=0; runs INTERN ASSIGN CronEd.CA.Profile[31]:=(CronEd.CA_TPR)
rounded rectangle at (280,440)-(311,461): text "%d"; shows CronEd.CA.Profile[32]; invisible if CronEd.CA_DayL<32; alarm colour if CronEd.CA.Profile[32]=0; runs INTERN ASSIGN CronEd.CA.Profile[32]:=(CronEd.CA_TPR)
rounded rectangle at (310,440)-(341,461): text "%d"; shows CronEd.CA.Profile[33]; invisible if CronEd.CA_DayL<33; alarm colour if CronEd.CA.Profile[33]=0; runs INTERN ASSIGN CronEd.CA.Profile[33]:=(CronEd.CA_TPR)
rounded rectangle at (340,440)-(371,461): text "%d"; shows CronEd.CA.Profile[34]; invisible if CronEd.CA_DayL<34; alarm colour if CronEd.CA.Profile[34]=0; runs INTERN ASSIGN CronEd.CA.Profile[34]:=(CronEd.CA_TPR)
rounded rectangle at (160,460)-(191,481): text "%d"; shows CronEd.CA.Profile[35]; invisible if CronEd.CA_DayL<35; alarm colour if CronEd.CA.Profile[35]=0; runs INTERN ASSIGN CronEd.CA.Profile[35]:=(CronEd.CA_TPR)
rectangle at (120,460)-(151,481): text "36"; invisible if CronEd.CA_DayL<35
rounded rectangle at (190,460)-(221,481): text "%d"; shows CronEd.CA.Profile[36]; invisible if CronEd.CA_DayL<36; alarm colour if CronEd.CA.Profile[36]=0; runs INTERN ASSIGN CronEd.CA.Profile[36]:=(CronEd.CA_TPR)
rounded rectangle at (220,460)-(251,481): text "%d"; shows CronEd.CA.Profile[37]; invisible if CronEd.CA_DayL<37; alarm colour if CronEd.CA.Profile[37]=0; runs INTERN ASSIGN CronEd.CA.Profile[37]:=(CronEd.CA_TPR)
rounded rectangle at (250,460)-(281,481): text "%d"; shows CronEd.CA.Profile[38]; invisible if CronEd.CA_DayL<38; alarm colour if CronEd.CA.Profile[38]=0; runs INTERN ASSIGN CronEd.CA.Profile[38]:=(CronEd.CA_TPR)
rounded rectangle at (280,460)-(311,481): text "%d"; shows CronEd.CA.Profile[39]; invisible if CronEd.CA_DayL<39; alarm colour if CronEd.CA.Profile[39]=0; runs INTERN ASSIGN CronEd.CA.Profile[39]:=(CronEd.CA_TPR)
rounded rectangle at (310,460)-(341,481): text "%d"; shows CronEd.CA.Profile[40]; invisible if CronEd.CA_DayL<40; alarm colour if CronEd.CA.Profile[40]=0; runs INTERN ASSIGN CronEd.CA.Profile[40]:=(CronEd.CA_TPR)
rounded rectangle at (340,460)-(371,481): text "%d"; shows CronEd.CA.Profile[41]; invisible if CronEd.CA_DayL<41; alarm colour if CronEd.CA.Profile[41]=0; runs INTERN ASSIGN CronEd.CA.Profile[41]:=(CronEd.CA_TPR)
rectangle at (310,60)-(371,81): text "Year"
rectangle at (370,60)-(411,81): text "%d"; shows CronEd.CN_YSel; alarm colour if CronEd.CN_YSel<>CronEd.CN_YAct; editable 2000..2100
rectangle at (480,60)-(761,81): text "%s"; shows CronEd.Message
button at (10,50)-(71,81): text "REINIT"; runs INTERN ASSIGN CRON03.InitOK:=(FALSE);INTERN ASSIGN CRON04.InitOK:=(FALSE);INTERN ASSIGN CRON05.InitOK:=(FALSE);INTERN ASSIGN CRON06.InitOK:=(FALSE);INTERN ASSIGN CRON01.InitOK:=(FALSE)
2 more shapes without text or variables
*)

(* Visualisation VIS_VRD01
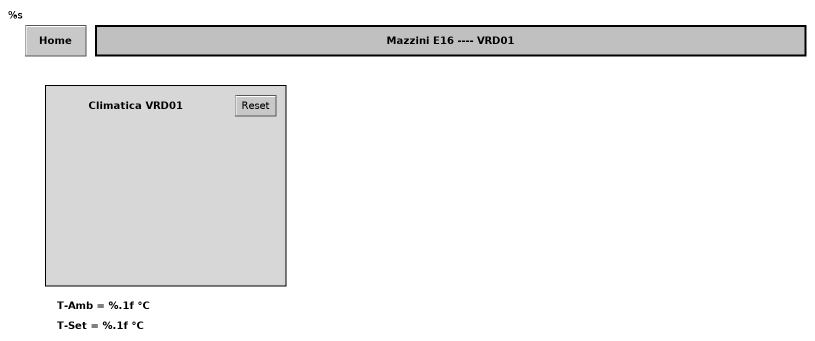
rectangle at (0,0)-(0,0): text "%s"; shows VRD01_Clima.Points[INDEX].X; invisible if INDEX>4; editable
rectangle at (0,0)-(0,0): text "%s"; shows VRD01_Clima.Points[INDEX].Y; invisible if INDEX>4; editable
rectangle at (40,80)-(201,101): text "Climatica VRD01"
button at (220,80)-(261,101): text "Reset"; runs INTERN ASSIGN VRD01_Clima.InitOK:=(FALSE)
button at (10,10)-(71,41): text "Home"; opens PLC_VISU
rectangle at (40,300)-(181,321): text "T-Set = %.1f °C"; shows INT_TO_REAL(.VRD01.Ctrl_SetPoint)/10
rectangle at (40,280)-(181,301): text "T-Amb = %.1f °C"; shows INT_TO_REAL(.T_AMB)/10; alarm colour if T_AMB>2000
rectangle at (80,10)-(791,41): text "Mazzini E16 ---- VRD01"
1 more shapes without text or variables
*)

(* Visualisation VIS_VRD02
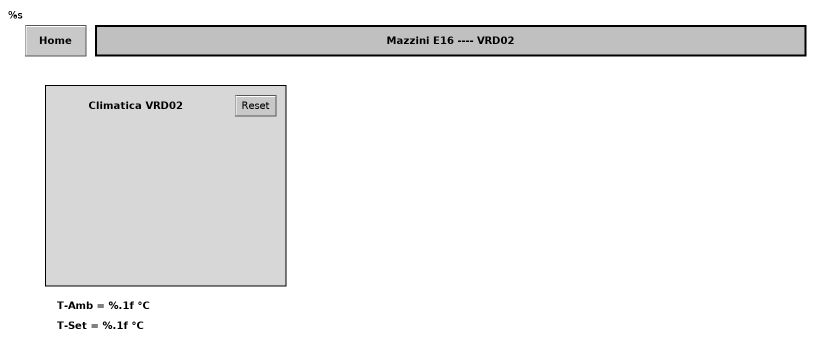
rectangle at (0,0)-(0,0): text "%s"; shows VRD01_Clima.Points[INDEX].X; invisible if INDEX>4; editable
rectangle at (0,0)-(0,0): text "%s"; shows VRD01_Clima.Points[INDEX].Y; invisible if INDEX>4; editable
rectangle at (40,80)-(201,101): text "Climatica VRD02"
button at (220,80)-(261,101): text "Reset"; runs INTERN ASSIGN VRD02_Clima.InitOK:=(FALSE)
button at (10,10)-(71,41): text "Home"; opens PLC_VISU
rectangle at (40,300)-(181,321): text "T-Set = %.1f °C"; shows INT_TO_REAL(.VRD02.Ctrl_SetPoint)/10
rectangle at (40,280)-(181,301): text "T-Amb = %.1f °C"; shows INT_TO_REAL(.T_AMB)/10; alarm colour if T_AMB>2000
rectangle at (80,10)-(791,41): text "Mazzini E16 ---- VRD02"
1 more shapes without text or variables
*)

(* Visualisation VIS_VRD03
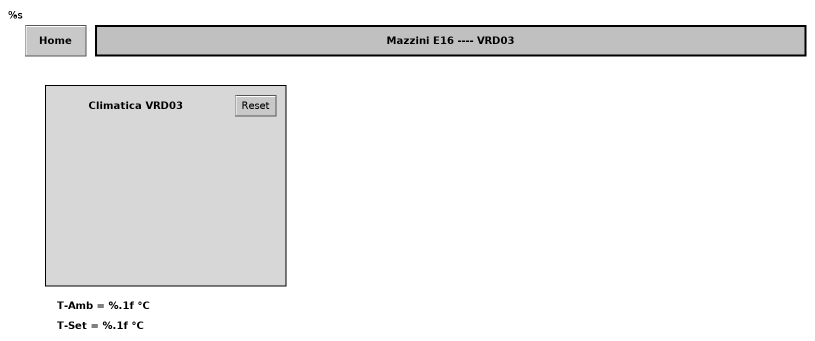
rectangle at (0,0)-(0,0): text "%s"; shows VRD01_Clima.Points[INDEX].X; invisible if INDEX>4; editable
rectangle at (0,0)-(0,0): text "%s"; shows VRD01_Clima.Points[INDEX].Y; invisible if INDEX>4; editable
rectangle at (40,80)-(201,101): text "Climatica VRD03"
button at (220,80)-(261,101): text "Reset"; runs INTERN ASSIGN VRD03_Clima.InitOK:=(FALSE)
button at (10,10)-(71,41): text "Home"; opens PLC_VISU
rectangle at (40,300)-(181,321): text "T-Set = %.1f °C"; shows INT_TO_REAL(.VRD03.Ctrl_SetPoint)/10
rectangle at (40,280)-(181,301): text "T-Amb = %.1f °C"; shows INT_TO_REAL(.T_AMB)/10; alarm colour if T_AMB>2000
rectangle at (80,10)-(791,41): text "Mazzini E16 ---- VRD03"
1 more shapes without text or variables
*)
